// SIMATIC STEP 7 (V5.x) project e121001V002
// CPU: CPU 313C-2 DP
// CPU: CPU 313C-2 DP
// station: P_ADR_BUS
// station: Hardware
// station: OLD
// station: P_ADR_BUS
// station: Hardware
// station: SIMATIC 300(2)
// program: Programa S7(1)
// program: Programa S7(2)

SYMBOL_TABLE
"COUNT"	SFB 47	SFB 47	// Common counter module
"VAT_1"	VAT 1	
END_SYMBOL_TABLE

FUNCTION_BLOCK FB 30
VERSION : 0.1
BEGIN
// (block stored without names or comments; labels and parameter names are numbered)
NETWORK
TITLE =
      A     M 251.0;
      =     L 16.0;
      A     L 16.0;
      JNB   M001;
      L     DIW [AR2,P#26.0];
      L     DIW [AR2,P#4.0];
      +I;
      T     DIW [AR2,P#28.0];
M001: NOP   0;
      A     L 16.0;
      A(;
      A(;
      L     DID [AR2,P#0.0];
      L     DIW [AR2,P#26.0];
      >=I;
      );
      A(;
      L     DID [AR2,P#0.0];
      L     DIW [AR2,P#36.0];
      <I;
      );
      O;
      A(;
      L     DID [AR2,P#0.0];
      L     DIW [AR2,P#26.0];
      >=I;
      );
      A(;
      L     DID [AR2,P#0.0];
      L     DIW [AR2,P#28.0];
      <I;
      );
      );
      =     DIX [AR2,P#16.0];
NETWORK
TITLE =
      A     DIX [AR2,P#16.0];
      =     L 16.0;
      A     L 16.0;
      JNB   M002;
      L     DIW [AR2,P#34.0];
      L     164;
      *I;
      T     DIW [AR2,P#14.0];
M002: NOP   0;
      A     L 16.0;
      JNB   M003;
      L     0;
      T     DIW [AR2,P#18.0];
M003: NOP   0;
NETWORK
TITLE =
      A     M 251.0;
      =     L 16.0;
      A     L 16.0;
      JNB   M004;
      L     DIW [AR2,P#36.0];
      L     DIW [AR2,P#4.0];
      +I;
      T     DIW [AR2,P#38.0];
M004: NOP   0;
      A     L 16.0;
      A(;
      A(;
      L     DID [AR2,P#0.0];
      L     DIW [AR2,P#36.0];
      >=I;
      );
      A(;
      L     DID [AR2,P#0.0];
      L     DIW [AR2,P#46.0];
      <I;
      );
      O;
      A(;
      L     DID [AR2,P#0.0];
      L     DIW [AR2,P#36.0];
      >=I;
      );
      A(;
      L     DID [AR2,P#0.0];
      L     DIW [AR2,P#38.0];
      <I;
      );
      );
      =     DIX [AR2,P#16.1];
NETWORK
TITLE =
      A     DIX [AR2,P#16.1];
      =     L 16.0;
      A     L 16.0;
      AN    T 13;
      =     L 16.1;
      A     L 16.1;
      JNB   M005;
      L     DIW [AR2,P#44.0];
      L     164;
      *I;
      T     DIW [AR2,P#14.0];
M005: NOP   0;
      A     L 16.1;
      JNB   M006;
      L     1;
      T     DIW [AR2,P#18.0];
M006: NOP   0;
      A     L 16.0;
      A     T 13;
      =     L 16.1;
      A     L 16.1;
      JNB   M007;
      L     80;
      L     164;
      *I;
      T     DIW [AR2,P#14.0];
M007: NOP   0;
      A     L 16.1;
      JNB   M008;
      L     1;
      T     DIW [AR2,P#18.0];
M008: NOP   0;
NETWORK
TITLE =
      A     M 251.0;
      =     L 16.0;
      A     L 16.0;
      JNB   M009;
      L     DIW [AR2,P#46.0];
      L     DIW [AR2,P#4.0];
      +I;
      T     DIW [AR2,P#48.0];
M009: NOP   0;
      A     L 16.0;
      A(;
      A(;
      L     DID [AR2,P#0.0];
      L     DIW [AR2,P#46.0];
      >=I;
      );
      A(;
      L     DID [AR2,P#0.0];
      L     DIW [AR2,P#56.0];
      <I;
      );
      O;
      A(;
      L     DID [AR2,P#0.0];
      L     DIW [AR2,P#46.0];
      >=I;
      );
      A(;
      L     DID [AR2,P#0.0];
      L     DIW [AR2,P#48.0];
      <I;
      );
      );
      =     DIX [AR2,P#16.2];
NETWORK
TITLE =
      A     DIX [AR2,P#16.2];
      =     L 16.0;
      A     L 16.0;
      AN    T 13;
      =     L 16.1;
      A     L 16.1;
      JNB   M010;
      L     DIW [AR2,P#54.0];
      L     164;
      *I;
      T     DIW [AR2,P#14.0];
M010: NOP   0;
      A     L 16.1;
      JNB   M011;
      L     2;
      T     DIW [AR2,P#18.0];
M011: NOP   0;
      A     L 16.0;
      A     T 13;
      =     L 16.1;
      A     L 16.1;
      JNB   M012;
      L     80;
      L     164;
      *I;
      T     DIW [AR2,P#14.0];
M012: NOP   0;
      A     L 16.1;
      JNB   M013;
      L     1;
      T     DIW [AR2,P#18.0];
M013: NOP   0;
NETWORK
TITLE =
      A     M 251.0;
      =     L 16.0;
      A     L 16.0;
      JNB   M014;
      L     DIW [AR2,P#56.0];
      L     DIW [AR2,P#4.0];
      +I;
      T     DIW [AR2,P#58.0];
M014: NOP   0;
      A     L 16.0;
      A(;
      A(;
      L     DID [AR2,P#0.0];
      L     DIW [AR2,P#56.0];
      >=I;
      );
      A(;
      L     DID [AR2,P#0.0];
      L     DIW [AR2,P#66.0];
      <I;
      );
      O;
      A(;
      L     DID [AR2,P#0.0];
      L     DIW [AR2,P#56.0];
      >=I;
      );
      A(;
      L     DID [AR2,P#0.0];
      L     DIW [AR2,P#58.0];
      <I;
      );
      );
      =     DIX [AR2,P#16.3];
NETWORK
TITLE =
      A     DIX [AR2,P#16.3];
      =     L 16.0;
      A     L 16.0;
      AN    T 13;
      =     L 16.1;
      A     L 16.1;
      JNB   M015;
      L     DIW [AR2,P#64.0];
      L     164;
      *I;
      T     DIW [AR2,P#14.0];
M015: NOP   0;
      A     L 16.1;
      JNB   M016;
      L     3;
      T     DIW [AR2,P#18.0];
M016: NOP   0;
      A     L 16.0;
      A     T 13;
      =     L 16.1;
      A     L 16.1;
      JNB   M017;
      L     80;
      L     164;
      *I;
      T     DIW [AR2,P#14.0];
M017: NOP   0;
      A     L 16.1;
      JNB   M018;
      L     3;
      T     DIW [AR2,P#18.0];
M018: NOP   0;
NETWORK
TITLE =
      A     M 251.0;
      =     L 16.0;
      A     L 16.0;
      JNB   M019;
      L     DIW [AR2,P#66.0];
      L     DIW [AR2,P#4.0];
      +I;
      T     DIW [AR2,P#68.0];
M019: NOP   0;
      A     L 16.0;
      A(;
      A(;
      L     DID [AR2,P#0.0];
      L     DIW [AR2,P#66.0];
      >=I;
      );
      A(;
      L     DID [AR2,P#0.0];
      L     DIW [AR2,P#76.0];
      <I;
      );
      O;
      A(;
      L     DID [AR2,P#0.0];
      L     DIW [AR2,P#66.0];
      >=I;
      );
      A(;
      L     DID [AR2,P#0.0];
      L     DIW [AR2,P#68.0];
      <I;
      );
      );
      =     DIX [AR2,P#16.4];
NETWORK
TITLE =
      A     DIX [AR2,P#16.4];
      =     L 16.0;
      A     L 16.0;
      AN    T 13;
      =     L 16.1;
      A     L 16.1;
      JNB   M020;
      L     DIW [AR2,P#74.0];
      L     164;
      *I;
      T     DIW [AR2,P#14.0];
M020: NOP   0;
      A     L 16.1;
      JNB   M021;
      L     4;
      T     DIW [AR2,P#18.0];
M021: NOP   0;
      A     L 16.0;
      A     T 13;
      =     L 16.1;
      A     L 16.1;
      JNB   M022;
      L     80;
      L     164;
      *I;
      T     DIW [AR2,P#14.0];
M022: NOP   0;
      A     L 16.1;
      JNB   M023;
      L     4;
      T     DIW [AR2,P#18.0];
M023: NOP   0;
NETWORK
TITLE =
      A     M 251.0;
      =     L 16.0;
      A     L 16.0;
      JNB   M024;
      L     DIW [AR2,P#76.0];
      L     DIW [AR2,P#4.0];
      +I;
      T     DIW [AR2,P#78.0];
M024: NOP   0;
      A     L 16.0;
      A(;
      A(;
      L     DID [AR2,P#0.0];
      L     DIW [AR2,P#76.0];
      >=I;
      );
      A(;
      L     DID [AR2,P#0.0];
      L     DIW [AR2,P#86.0];
      <I;
      );
      O;
      A(;
      L     DID [AR2,P#0.0];
      L     DIW [AR2,P#76.0];
      >=I;
      );
      A(;
      L     DID [AR2,P#0.0];
      L     DIW [AR2,P#78.0];
      <I;
      );
      );
      =     DIX [AR2,P#16.5];
NETWORK
TITLE =
      A     DIX [AR2,P#16.5];
      =     L 16.0;
      A     L 16.0;
      AN    T 13;
      =     L 16.1;
      A     L 16.1;
      JNB   M025;
      L     DIW [AR2,P#84.0];
      L     164;
      *I;
      T     DIW [AR2,P#14.0];
M025: NOP   0;
      A     L 16.1;
      JNB   M026;
      L     5;
      T     DIW [AR2,P#18.0];
M026: NOP   0;
      A     L 16.0;
      A     T 13;
      =     L 16.1;
      A     L 16.1;
      JNB   M027;
      L     80;
      L     164;
      *I;
      T     DIW [AR2,P#14.0];
M027: NOP   0;
      A     L 16.1;
      JNB   M028;
      L     5;
      T     DIW [AR2,P#18.0];
M028: NOP   0;
NETWORK
TITLE =
      A     M 251.0;
      =     L 16.0;
      A     L 16.0;
      JNB   M029;
      L     DIW [AR2,P#86.0];
      L     DIW [AR2,P#4.0];
      +I;
      T     DIW [AR2,P#88.0];
M029: NOP   0;
      A     L 16.0;
      A(;
      A(;
      L     DID [AR2,P#0.0];
      L     DIW [AR2,P#86.0];
      >=I;
      );
      A(;
      L     DID [AR2,P#0.0];
      L     DIW [AR2,P#96.0];
      <I;
      );
      O;
      A(;
      L     DID [AR2,P#0.0];
      L     DIW [AR2,P#86.0];
      >=I;
      );
      A(;
      L     DID [AR2,P#0.0];
      L     DIW [AR2,P#88.0];
      <I;
      );
      );
      =     DIX [AR2,P#16.6];
NETWORK
TITLE =
      A     DIX [AR2,P#16.6];
      =     L 16.0;
      A     L 16.0;
      AN    T 13;
      =     L 16.1;
      A     L 16.1;
      JNB   M030;
      L     DIW [AR2,P#94.0];
      L     164;
      *I;
      T     DIW [AR2,P#14.0];
M030: NOP   0;
      A     L 16.1;
      JNB   M031;
      L     6;
      T     DIW [AR2,P#18.0];
M031: NOP   0;
      A     L 16.0;
      A     T 13;
      =     L 16.1;
      A     L 16.1;
      JNB   M032;
      L     80;
      L     164;
      *I;
      T     DIW [AR2,P#14.0];
M032: NOP   0;
      A     L 16.1;
      JNB   M033;
      L     6;
      T     DIW [AR2,P#18.0];
M033: NOP   0;
NETWORK
TITLE =
      A     M 251.0;
      =     L 16.0;
      A     L 16.0;
      JNB   M034;
      L     DIW [AR2,P#96.0];
      L     DIW [AR2,P#4.0];
      +I;
      T     DIW [AR2,P#98.0];
M034: NOP   0;
      A     L 16.0;
      A(;
      A(;
      L     DID [AR2,P#0.0];
      L     DIW [AR2,P#96.0];
      >=I;
      );
      A(;
      L     DID [AR2,P#0.0];
      L     DIW [AR2,P#106.0];
      <I;
      );
      O;
      A(;
      L     DID [AR2,P#0.0];
      L     DIW [AR2,P#96.0];
      >=I;
      );
      A(;
      L     DID [AR2,P#0.0];
      L     DIW [AR2,P#98.0];
      <I;
      );
      );
      =     DIX [AR2,P#16.7];
NETWORK
TITLE =
      A     DIX [AR2,P#16.7];
      =     L 16.0;
      A     L 16.0;
      AN    T 13;
      =     L 16.1;
      A     L 16.1;
      JNB   M035;
      L     DIW [AR2,P#104.0];
      L     164;
      *I;
      T     DIW [AR2,P#14.0];
M035: NOP   0;
      A     L 16.1;
      JNB   M036;
      L     7;
      T     DIW [AR2,P#18.0];
M036: NOP   0;
      A     L 16.0;
      A     T 13;
      =     L 16.1;
      A     L 16.1;
      JNB   M037;
      L     80;
      L     164;
      *I;
      T     DIW [AR2,P#14.0];
M037: NOP   0;
      A     L 16.1;
      JNB   M038;
      L     7;
      T     DIW [AR2,P#18.0];
M038: NOP   0;
NETWORK
TITLE =
      A     M 251.0;
      =     L 16.0;
      A     L 16.0;
      JNB   M039;
      L     DIW [AR2,P#106.0];
      L     DIW [AR2,P#4.0];
      +I;
      T     DIW [AR2,P#108.0];
M039: NOP   0;
      A     L 16.0;
      A(;
      L     DID [AR2,P#0.0];
      L     DIW [AR2,P#106.0];
      >=I;
      );
      A(;
      L     DID [AR2,P#0.0];
      L     DIW [AR2,P#108.0];
      <I;
      );
      =     DIX [AR2,P#17.0];
NETWORK
TITLE =
      A     DIX [AR2,P#17.0];
      =     L 16.0;
      A     L 16.0;
      JNB   M040;
      L     DIW [AR2,P#114.0];
      L     164;
      *I;
      T     DIW [AR2,P#14.0];
M040: NOP   0;
      A     L 16.0;
      JNB   M041;
      L     8;
      T     DIW [AR2,P#18.0];
M041: NOP   0;
NETWORK
TITLE =
      A     DIX [AR2,P#8.0];
      =     L 26.0;
      A     L 26.0;
      JNB   M042;
      L     DIW [AR2,P#6.0];
      L     5;
      *I;
      T     LW 2;
M042: NOP   0;
      A     L 26.0;
      JNB   M043;
      L     LW 2;
      L     13;
      +I;
      T     LW 4;
M043: NOP   0;
      A     L 26.0;
      JNB   M044;
      CALL  FC 103 (
           $1                       := 30,
           $2                       := 1,
           $3                       := 1,
           $4                       := 30,
           $5                       := P#L 4.0);
M044: NOP   0;
      A     L 26.0;
      JNB   M045;
      L     LW 2;
      L     17;
      +I;
      T     LW 6;
M045: NOP   0;
      A     L 26.0;
      JNB   M046;
      CALL  FC 103 (
           $1                       := 30,
           $2                       := 12,
           $3                       := 12,
           $4                       := 30,
           $5                       := P#L 6.0);
M046: NOP   0;
      A     L 26.0;
      JNB   M047;
      L     DIW [AR2,P#22.0];
      L     100;
      +I;
      T     LW 0;
M047: NOP   0;
      A     L 26.0;
      JNB   M048;
      CALL  FC 103 (
           $1                       := 30,
           $2                       := 13,
           $3                       := 92,
           $4                       := P#L 0.0,
           $5                       := 2);
M048: NOP   0;
      A     L 26.0;
      BLD   102;
      R     DB30.DBX 8.0;
      A(;
      A     L 26.0;
      JNB   M049;
      L     DB30.DBW 6;
      L     1;
      +I;
      T     DB30.DBW 6;
      AN    OV;
      SAVE;
      CLR;
M049: A     BR;
      );
      A(;
      L     DB30.DBW 6;
      L     8;
      >I;
      );
      JNB   M050;
      L     8;
      T     DB30.DBW 6;
M050: NOP   0;
NETWORK
TITLE =
      A     DIX [AR2,P#8.1];
      =     L 26.0;
      A     L 26.0;
      JNB   M051;
      L     DIW [AR2,P#6.0];
      L     5;
      *I;
      T     LW 2;
M051: NOP   0;
      A     L 26.0;
      JNB   M052;
      L     LW 2;
      L     17;
      +I;
      T     LW 4;
M052: NOP   0;
      A     L 26.0;
      JNB   M053;
      CALL  FC 103 (
           $1                       := 30,
           $2                       := 12,
           $3                       := 12,
           $4                       := 30,
           $5                       := P#L 4.0);
M053: NOP   0;
      A     L 26.0;
      JNB   M054;
      L     DIW [AR2,P#22.0];
      L     100;
      +I;
      T     LW 0;
M054: NOP   0;
      A     L 26.0;
      JNB   M055;
      CALL  FC 103 (
           $1                       := 30,
           $2                       := 13,
           $3                       := 92,
           $4                       := P#L 0.0,
           $5                       := 2);
M055: NOP   0;
      A     L 26.0;
      BLD   102;
      R     DB30.DBX 8.1;
NETWORK
TITLE =
      A     DIX [AR2,P#8.4];
      =     L 26.0;
      A     L 26.0;
      JNB   M056;
      L     DIW [AR2,P#22.0];
      L     100;
      +I;
      T     LW 0;
M056: NOP   0;
      A     L 26.0;
      JNB   M057;
      CALL  FC 103 (
           $1                       := 30,
           $2                       := 13,
           $3                       := 92,
           $4                       := P#L 0.0,
           $5                       := 2);
M057: NOP   0;
      A     L 26.0;
      BLD   102;
      R     M 4.0;
NETWORK
TITLE =
      A     DIX [AR2,P#8.5];
      =     L 26.0;
      A     L 26.0;
      JNB   M058;
      L     DB1.DBW 42;
      L     100;
      +I;
      T     LW 8;
M058: NOP   0;
      A     L 26.0;
      JNB   M059;
      CALL  FC 103 (
           $1                       := 121,
           $2                       := 2,
           $3                       := 92,
           $4                       := P#L 8.0,
           $5                       := 2);
M059: NOP   0;
      A     L 26.0;
      BLD   102;
      R     M 4.2;
NETWORK
TITLE =
      A     DIX [AR2,P#8.3];
      =     L 26.0;
      A     L 26.0;
      JNB   M060;
      L     DB1.DBW 38;
      L     100;
      +I;
      T     LW 10;
M060: NOP   0;
      A     L 26.0;
      JNB   M061;
      L     DB1.DBW 40;
      L     100;
      +I;
      T     LW 12;
M061: NOP   0;
      A     L 26.0;
      JNB   M062;
      CALL  FC 103 (
           $1                       := P#L 10.0,
           $2                       := 2,
           $3                       := 92,
           $4                       := P#L 12.0,
           $5                       := 2);
M062: NOP   0;
      A     L 26.0;
      BLD   102;
      R     M 4.1;
NETWORK
TITLE =
      A     DIX [AR2,P#8.6];
      =     L 26.0;
      A     L 26.0;
      JNB   M063;
      L     DB1.DBW 12;
      L     77;
      +I;
      T     LW 14;
M063: NOP   0;
      A     L 26.0;
      JNB   M064;
      CALL  FC 103 (
           $1                       := 30,
           $2                       := 6,
           $3                       := 6,
           $4                       := 30,
           $5                       := P#L 14.0);
M064: NOP   0;
      A     L 26.0;
      JNB   M065;
      L     DIW [AR2,P#22.0];
      L     100;
      +I;
      T     LW 0;
M065: NOP   0;
      A     L 26.0;
      JNB   M066;
      CALL  FC 103 (
           $1                       := 30,
           $2                       := 13,
           $3                       := 92,
           $4                       := P#L 0.0,
           $5                       := 2);
M066: NOP   0;
      A     L 26.0;
      BLD   102;
      R     DB30.DBX 8.6;
      A(;
      A     L 26.0;
      JNB   M067;
      L     DB1.DBW 12;
      L     1;
      +I;
      T     DB1.DBW 12;
      AN    OV;
      SAVE;
      CLR;
M067: A     BR;
      );
      A(;
      L     DB1.DBW 12;
      L     3;
      >I;
      );
      JNB   M068;
      L     3;
      T     DB1.DBW 12;
M068: NOP   0;
NETWORK
TITLE =
      A     M 251.0;
      =     L 26.0;
      A     L 26.0;
      JNB   M069;
      L     DIW [AR2,P#154.0];
      L     10;
      +I;
      T     DIW [AR2,P#166.0];
M069: NOP   0;
      A     L 26.0;
      JNB   M070;
      L     DIW [AR2,P#154.0];
      L     10;
      -I;
      T     DIW [AR2,P#168.0];
M070: NOP   0;
      A     L 26.0;
      A(;
      L     DIW [AR2,P#12.0];
      L     DIW [AR2,P#168.0];
      >=I;
      );
      A(;
      L     DIW [AR2,P#12.0];
      L     DIW [AR2,P#166.0];
      <=I;
      );
      =     DIX [AR2,P#20.0];
NETWORK
TITLE =
      A     M 251.0;
      =     L 26.0;
      A     L 26.0;
      JNB   M071;
      L     DIW [AR2,P#156.0];
      L     10;
      +I;
      T     DIW [AR2,P#170.0];
M071: NOP   0;
      A     L 26.0;
      JNB   M072;
      L     DIW [AR2,P#156.0];
      L     10;
      -I;
      T     LW 16;
M072: NOP   0;
      A     L 26.0;
      A(;
      L     DIW [AR2,P#12.0];
      L     LW 16;
      >=I;
      );
      A(;
      L     DIW [AR2,P#12.0];
      L     DIW [AR2,P#170.0];
      <=I;
      );
      =     DIX [AR2,P#20.1];
NETWORK
TITLE =
      A     M 251.0;
      =     L 26.0;
      A     L 26.0;
      JNB   M073;
      L     DIW [AR2,P#158.0];
      L     10;
      +I;
      T     LW 18;
M073: NOP   0;
      A     L 26.0;
      JNB   M074;
      L     DIW [AR2,P#158.0];
      L     10;
      -I;
      T     LW 20;
M074: NOP   0;
      A     L 26.0;
      A(;
      L     DIW [AR2,P#12.0];
      L     LW 20;
      >=I;
      );
      A(;
      L     DIW [AR2,P#12.0];
      L     LW 18;
      <=I;
      );
      =     DIX [AR2,P#20.2];
NETWORK
TITLE =
      A     M 251.0;
      =     L 26.0;
      A     L 26.0;
      JNB   M075;
      L     DIW [AR2,P#160.0];
      L     10;
      +I;
      T     LW 22;
M075: NOP   0;
      A     L 26.0;
      JNB   M076;
      L     DIW [AR2,P#160.0];
      L     10;
      -I;
      T     LW 24;
M076: NOP   0;
      A     L 26.0;
      A(;
      L     DIW [AR2,P#12.0];
      L     LW 24;
      >=I;
      );
      A(;
      L     DIW [AR2,P#12.0];
      L     LW 22;
      <=I;
      );
      =     DIX [AR2,P#20.3];
NETWORK
TITLE =
      A     M 80.0;
      A     DIX [AR2,P#20.0];
      =     M 6.5;
END_FUNCTION_BLOCK

FUNCTION_BLOCK FB 50
VERSION : 0.1
BEGIN
// (block stored without names or comments; labels and parameter names are numbered)
NETWORK
TITLE =
END_FUNCTION_BLOCK

FUNCTION_BLOCK FB 51
VERSION : 0.1
BEGIN
// (block stored without names or comments; labels and parameter names are numbered)
NETWORK
TITLE =
END_FUNCTION_BLOCK

FUNCTION FC 1 : VOID
VERSION : 0.1
BEGIN
// (block stored without names or comments; labels and parameter names are numbered)
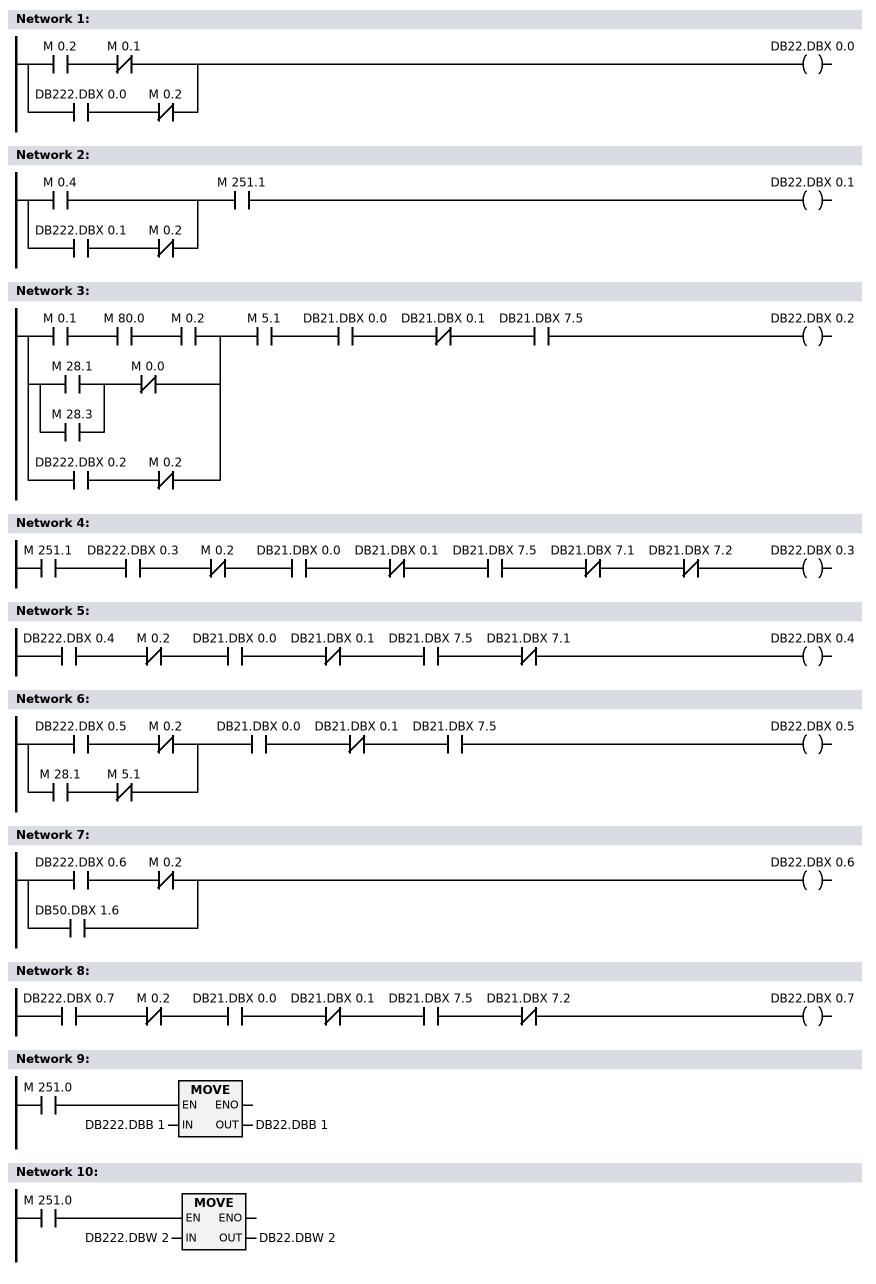
NETWORK
TITLE =
      A     M 0.2;
      AN    M 0.1;
      O;
      A     DB222.DBX 0.0;
      AN    M 0.2;
      =     DB22.DBX 0.0;
NETWORK
TITLE =
      A(;
      O     M 0.4;
      O;
      A     DB222.DBX 0.1;
      AN    M 0.2;
      );
      A     M 251.1;
      =     DB22.DBX 0.1;
NETWORK
TITLE =
      A(;
      A     M 0.1;
      A     M 80.0;
      A     M 0.2;
      O;
      A(;
      O     M 28.1;
      O     M 28.3;
      );
      AN    M 0.0;
      O;
      A     DB222.DBX 0.2;
      AN    M 0.2;
      );
      A     M 5.1;
      A     DB21.DBX 0.0;
      AN    DB21.DBX 0.1;
      A     DB21.DBX 7.5;
      =     DB22.DBX 0.2;
NETWORK
TITLE =
      A     M 251.1;
      A     DB222.DBX 0.3;
      AN    M 0.2;
      A     DB21.DBX 0.0;
      AN    DB21.DBX 0.1;
      A     DB21.DBX 7.5;
      AN    DB21.DBX 7.1;
      AN    DB21.DBX 7.2;
      =     DB22.DBX 0.3;
NETWORK
TITLE =
      A     DB222.DBX 0.4;
      AN    M 0.2;
      A     DB21.DBX 0.0;
      AN    DB21.DBX 0.1;
      A     DB21.DBX 7.5;
      AN    DB21.DBX 7.1;
      =     DB22.DBX 0.4;
NETWORK
TITLE =
      A(;
      A     DB222.DBX 0.5;
      AN    M 0.2;
      O;
      A     M 28.1;
      AN    M 5.1;
      );
      A     DB21.DBX 0.0;
      AN    DB21.DBX 0.1;
      A     DB21.DBX 7.5;
      =     DB22.DBX 0.5;
NETWORK
TITLE =
      A     DB222.DBX 0.6;
      AN    M 0.2;
      O     DB50.DBX 1.6;
      =     DB22.DBX 0.6;
NETWORK
TITLE =
      A     DB222.DBX 0.7;
      AN    M 0.2;
      A     DB21.DBX 0.0;
      AN    DB21.DBX 0.1;
      A     DB21.DBX 7.5;
      AN    DB21.DBX 7.2;
      =     DB22.DBX 0.7;
NETWORK
TITLE =
      A     M 251.0;
      JNB   M001;
      L     DB222.DBB 1;
      T     DB22.DBB 1;
M001: NOP   0;
NETWORK
TITLE =
      A     M 251.0;
      JNB   M002;
      L     DB222.DBW 2;
      T     DB22.DBW 2;
M002: NOP   0;
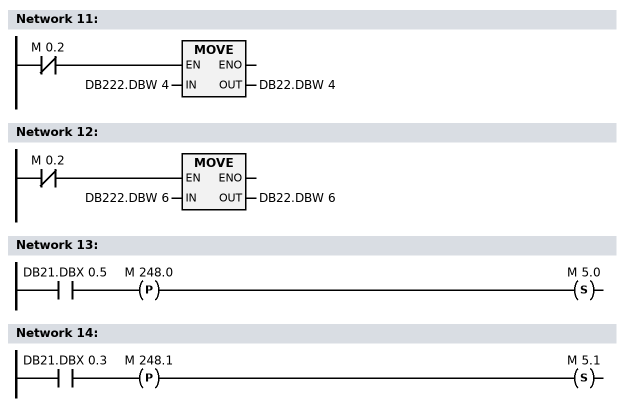
NETWORK
TITLE =
      AN    M 0.2;
      JNB   M003;
      L     DB222.DBW 4;
      T     DB22.DBW 4;
M003: NOP   0;
NETWORK
TITLE =
      AN    M 0.2;
      JNB   M004;
      L     DB222.DBW 6;
      T     DB22.DBW 6;
M004: NOP   0;
NETWORK
TITLE =
      A     DB21.DBX 0.5;
      FP    M 248.0;
      S     M 5.0;
NETWORK
TITLE =
      A     DB21.DBX 0.3;
      FP    M 248.1;
      S     M 5.1;
END_FUNCTION

FUNCTION FC 10 : VOID
VERSION : 0.1
VAR_TEMP
  TEMP0 : INT ;
END_VAR
BEGIN
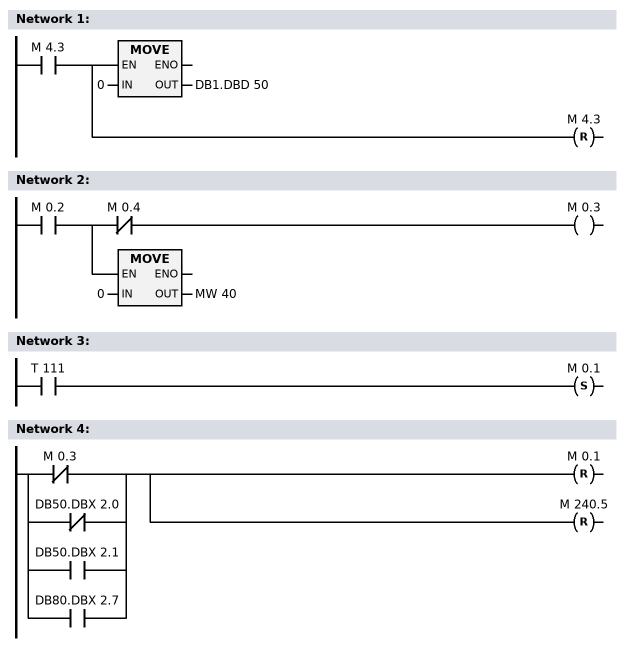
NETWORK
TITLE =
      A     M 4.3;
      =     L 2.0;
      A     L 2.0;
      JNB   _001;
      L     0;
      T     DB1.DBD 50;
_001: NOP   0;
      A     L 2.0;
      BLD   102;
      R     M 4.3;
NETWORK
TITLE =
      A     M 0.2;
      =     L 2.0;
      A     L 2.0;
      AN    M 0.4;
      =     M 0.3;
      A     L 2.0;
      JNB   _002;
      L     0;
      T     MW 40;
_002: NOP   0;
NETWORK
TITLE =
      A     T 111;
      S     M 0.1;
NETWORK
TITLE =
      ON    M 0.3;
      ON    DB50.DBX 2.0;
      O     DB50.DBX 2.1;
      O     DB80.DBX 2.7;
      R     M 0.1;
      R     M 240.5;
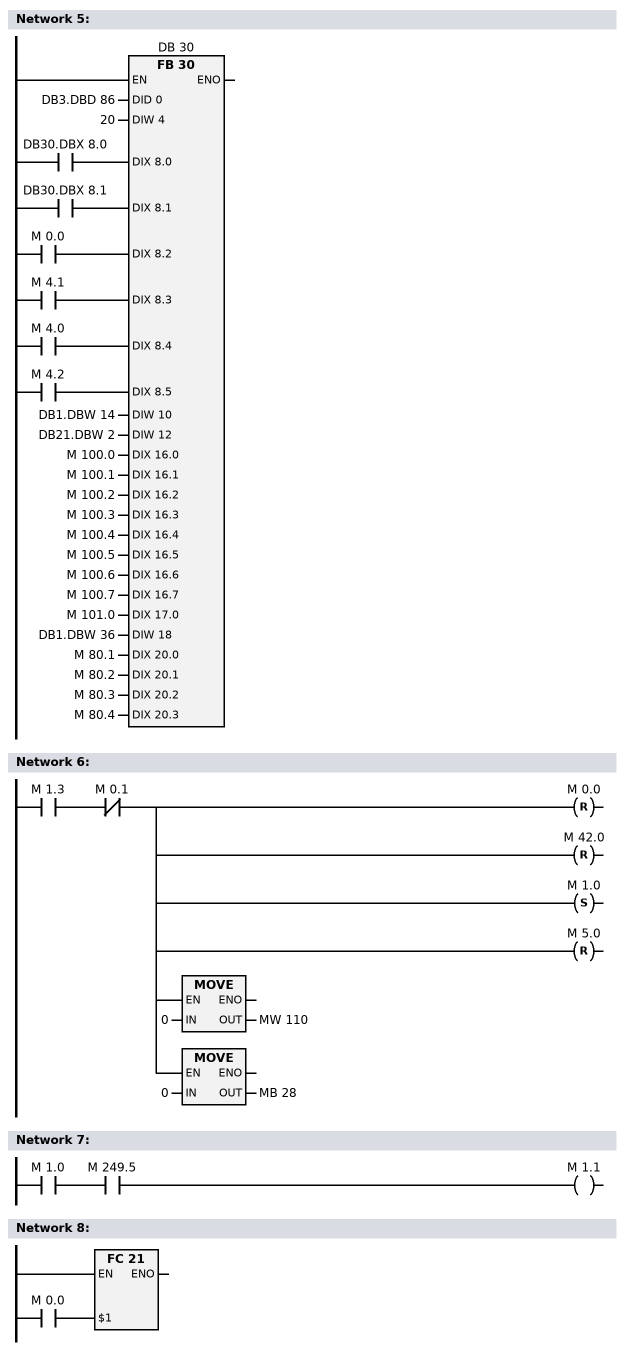
NETWORK
TITLE =
      A     DB30.DBX 8.0;
      =     L 2.0;
      BLD   103;
      A     DB30.DBX 8.1;
      =     L 2.1;
      BLD   103;
      A     M 0.0;
      =     L 2.2;
      BLD   103;
      A     M 4.1;
      =     L 2.3;
      BLD   103;
      A     M 4.0;
      =     L 2.4;
      BLD   103;
      A     M 4.2;
      =     L 2.5;
      BLD   103;
      CALL  FB 30 , DB 30 (
           DID 0                    := DB3.DBD 86,
           DIW 4                    := 20,
           DIX 8.0                  := L 2.0,
           DIX 8.1                  := L 2.1,
           DIX 8.2                  := L 2.2,
           DIX 8.3                  := L 2.3,
           DIX 8.4                  := L 2.4,
           DIX 8.5                  := L 2.5,
           DIW 10                   := DB1.DBW 14,
           DIW 12                   := DB21.DBW 2,
           DIX 16.0                 := M 100.0,
           DIX 16.1                 := M 100.1,
           DIX 16.2                 := M 100.2,
           DIX 16.3                 := M 100.3,
           DIX 16.4                 := M 100.4,
           DIX 16.5                 := M 100.5,
           DIX 16.6                 := M 100.6,
           DIX 16.7                 := M 100.7,
           DIX 17.0                 := M 101.0,
           DIW 18                   := DB1.DBW 36,
           DIX 20.0                 := M 80.1,
           DIX 20.1                 := M 80.2,
           DIX 20.2                 := M 80.3,
           DIX 20.3                 := M 80.4);
      NOP   0;
NETWORK
TITLE =
      A     M 1.3;
      AN    M 0.1;
      =     L 2.0;
      A     L 2.0;
      BLD   102;
      R     M 0.0;
      A     L 2.0;
      BLD   102;
      R     M 42.0;
      A     L 2.0;
      BLD   102;
      S     M 1.0;
      A     L 2.0;
      BLD   102;
      R     M 5.0;
      A     L 2.0;
      JNB   _003;
      L     0;
      T     MW 110;
_003: NOP   0;
      A     L 2.0;
      JNB   _004;
      L     0;
      T     MB 28;
_004: NOP   0;
NETWORK
TITLE =
      A     M 1.0;
      A     M 249.5;
      =     M 1.1;
NETWORK
TITLE =
      A     M 0.0;
      =     L 2.0;
      BLD   103;
      CALL  FC 21 (
           $1                       := L 2.0);
      NOP   0;
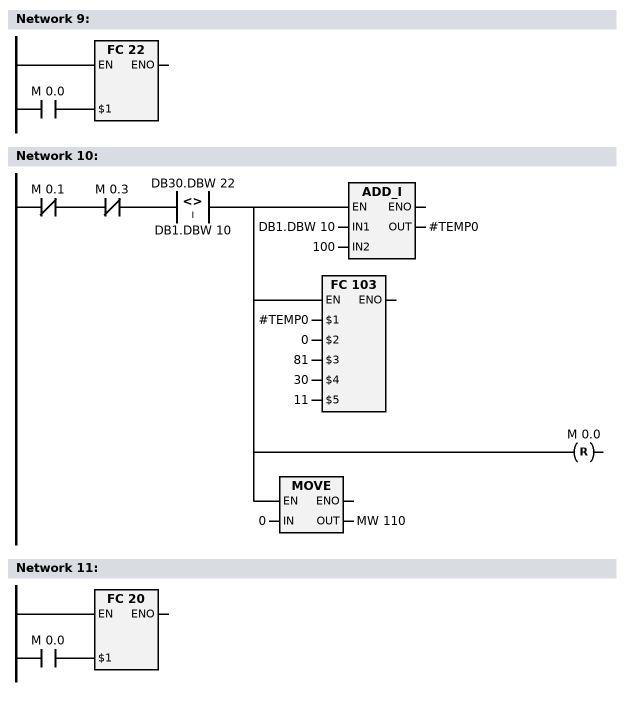
NETWORK
TITLE =
      A     M 0.0;
      =     L 2.0;
      BLD   103;
      CALL  FC 22 (
           $1                       := L 2.0);
      NOP   0;
NETWORK
TITLE =
      AN    M 0.1;
      AN    M 0.3;
      A(;
      L     DB30.DBW 22;
      L     DB1.DBW 10;
      <>I;
      );
      =     L 2.0;
      A     L 2.0;
      JNB   _005;
      L     DB1.DBW 10;
      L     100;
      +I;
      T     #TEMP0;
_005: NOP   0;
      A     L 2.0;
      JNB   _006;
      CALL  FC 103 (
           $1                       := #TEMP0,
           $2                       := 0,
           $3                       := 81,
           $4                       := 30,
           $5                       := 11);
_006: NOP   0;
      A     L 2.0;
      BLD   102;
      R     M 0.0;
      A     L 2.0;
      JNB   _007;
      L     0;
      T     MW 110;
_007: NOP   0;
NETWORK
TITLE =
      A     M 0.0;
      =     L 2.0;
      BLD   103;
      CALL  FC 20 (
           $1                       := L 2.0);
      NOP   0;
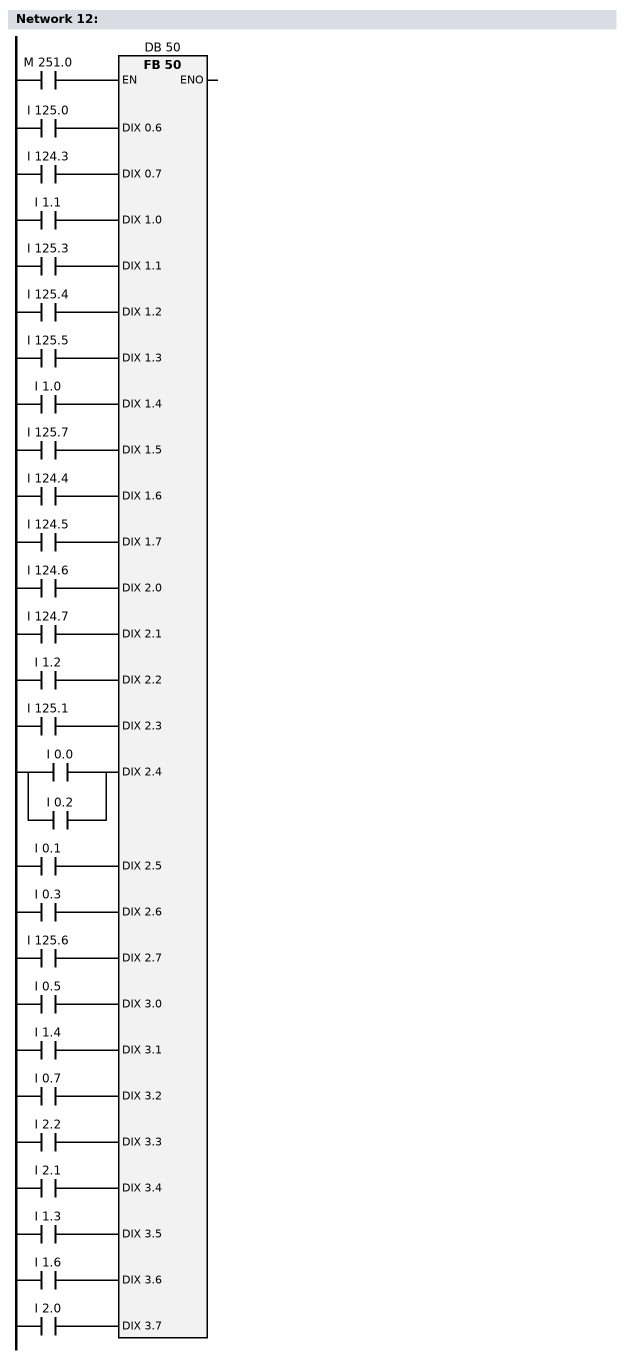
NETWORK
TITLE =
      A     I 125.0;
      =     L 2.6;
      BLD   103;
      A     I 124.3;
      =     L 2.7;
      BLD   103;
      A     I 1.1;
      =     L 3.0;
      BLD   103;
      A     I 125.3;
      =     L 3.1;
      BLD   103;
      A     I 125.4;
      =     L 3.2;
      BLD   103;
      A     I 125.5;
      =     L 3.3;
      BLD   103;
      A     I 1.0;
      =     L 3.4;
      BLD   103;
      A     I 125.7;
      =     L 3.5;
      BLD   103;
      A     I 124.4;
      =     L 3.6;
      BLD   103;
      A     I 124.5;
      =     L 3.7;
      BLD   103;
      A     I 124.6;
      =     L 4.0;
      BLD   103;
      A     I 124.7;
      =     L 4.1;
      BLD   103;
      A     I 1.2;
      =     L 4.2;
      BLD   103;
      A     I 125.1;
      =     L 4.3;
      BLD   103;
      A(;
      O     I 0.0;
      O     I 0.2;
      );
      =     L 4.4;
      BLD   103;
      A     I 0.1;
      =     L 4.5;
      BLD   103;
      A     I 0.3;
      =     L 4.6;
      BLD   103;
      A     I 125.6;
      =     L 4.7;
      BLD   103;
      A     I 0.5;
      =     L 5.0;
      BLD   103;
      A     I 1.4;
      =     L 5.1;
      BLD   103;
      A     I 0.7;
      =     L 5.2;
      BLD   103;
      A     I 2.2;
      =     L 5.3;
      BLD   103;
      A     I 2.1;
      =     L 5.4;
      BLD   103;
      A     I 1.3;
      =     L 5.5;
      BLD   103;
      A     I 1.6;
      =     L 5.6;
      BLD   103;
      A     I 2.0;
      =     L 5.7;
      BLD   103;
      A     M 251.0;
      JNB   _008;
      CALL  FB 50 , DB 50 (
           DIX 0.6                  := L 2.6,
           DIX 0.7                  := L 2.7,
           DIX 1.0                  := L 3.0,
           DIX 1.1                  := L 3.1,
           DIX 1.2                  := L 3.2,
           DIX 1.3                  := L 3.3,
           DIX 1.4                  := L 3.4,
           DIX 1.5                  := L 3.5,
           DIX 1.6                  := L 3.6,
           DIX 1.7                  := L 3.7,
           DIX 2.0                  := L 4.0,
           DIX 2.1                  := L 4.1,
           DIX 2.2                  := L 4.2,
           DIX 2.3                  := L 4.3,
           DIX 2.4                  := L 4.4,
           DIX 2.5                  := L 4.5,
           DIX 2.6                  := L 4.6,
           DIX 2.7                  := L 4.7,
           DIX 3.0                  := L 5.0,
           DIX 3.1                  := L 5.1,
           DIX 3.2                  := L 5.2,
           DIX 3.3                  := L 5.3,
           DIX 3.4                  := L 5.4,
           DIX 3.5                  := L 5.5,
           DIX 3.6                  := L 5.6,
           DIX 3.7                  := L 5.7);
_008: NOP   0;
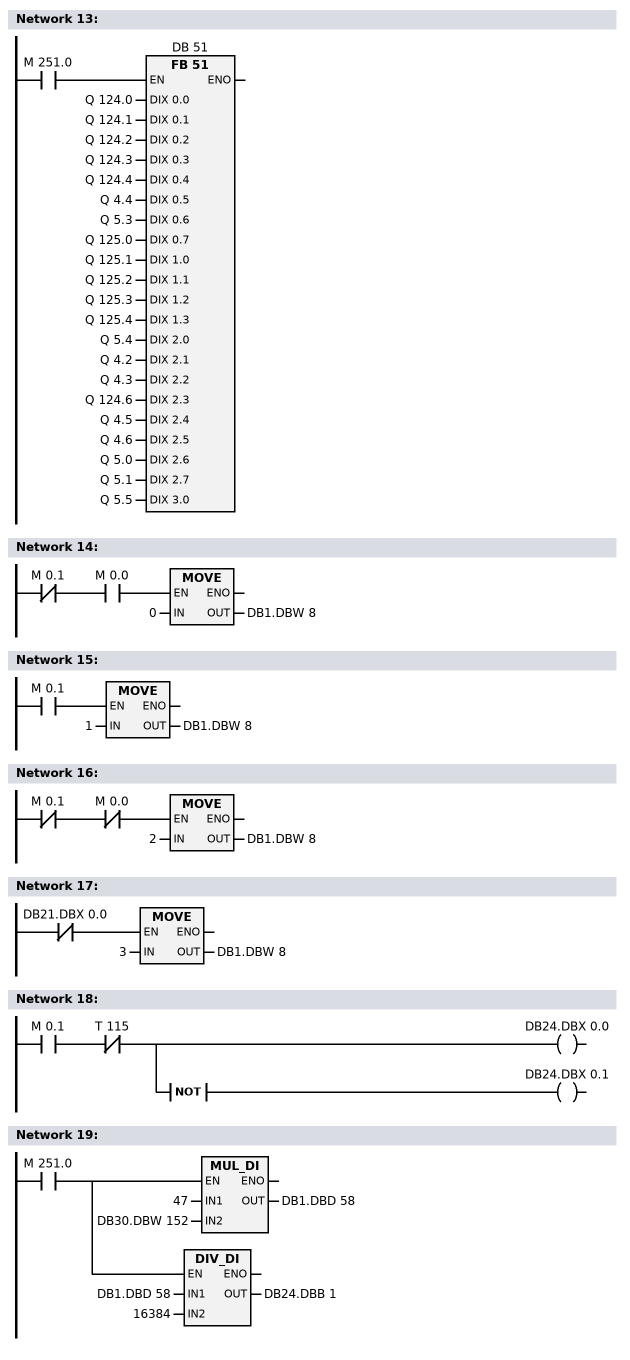
NETWORK
TITLE =
      A     M 251.0;
      JNB   _009;
      CALL  FB 51 , DB 51 (
           DIX 0.0                  := Q 124.0,
           DIX 0.1                  := Q 124.1,
           DIX 0.2                  := Q 124.2,
           DIX 0.3                  := Q 124.3,
           DIX 0.4                  := Q 124.4,
           DIX 0.5                  := Q 4.4,
           DIX 0.6                  := Q 5.3,
           DIX 0.7                  := Q 125.0,
           DIX 1.0                  := Q 125.1,
           DIX 1.1                  := Q 125.2,
           DIX 1.2                  := Q 125.3,
           DIX 1.3                  := Q 125.4,
           DIX 2.0                  := Q 5.4,
           DIX 2.1                  := Q 4.2,
           DIX 2.2                  := Q 4.3,
           DIX 2.3                  := Q 124.6,
           DIX 2.4                  := Q 4.5,
           DIX 2.5                  := Q 4.6,
           DIX 2.6                  := Q 5.0,
           DIX 2.7                  := Q 5.1,
           DIX 3.0                  := Q 5.5);
_009: NOP   0;
NETWORK
TITLE =
      AN    M 0.1;
      A     M 0.0;
      JNB   _00a;
      L     0;
      T     DB1.DBW 8;
_00a: NOP   0;
NETWORK
TITLE =
      A     M 0.1;
      JNB   _00b;
      L     1;
      T     DB1.DBW 8;
_00b: NOP   0;
NETWORK
TITLE =
      AN    M 0.1;
      AN    M 0.0;
      JNB   _00c;
      L     2;
      T     DB1.DBW 8;
_00c: NOP   0;
NETWORK
TITLE =
      AN    DB21.DBX 0.0;
      JNB   _00d;
      L     3;
      T     DB1.DBW 8;
_00d: NOP   0;
NETWORK
TITLE =
      A     M 0.1;
      AN    T 115;
      =     L 2.0;
      A     L 2.0;
      BLD   102;
      =     DB24.DBX 0.0;
      A     L 2.0;
      NOT;
      =     DB24.DBX 0.1;
NETWORK
TITLE =
      A     M 251.0;
      =     L 2.0;
      A     L 2.0;
      JNB   _00e;
      L     47;
      L     DB30.DBW 152;
      *D;
      T     DB1.DBD 58;
_00e: NOP   0;
      A     L 2.0;
      JNB   _00f;
      L     DB1.DBD 58;
      L     16384;
      /D;
      T     DB24.DBB 1;
_00f: NOP   0;
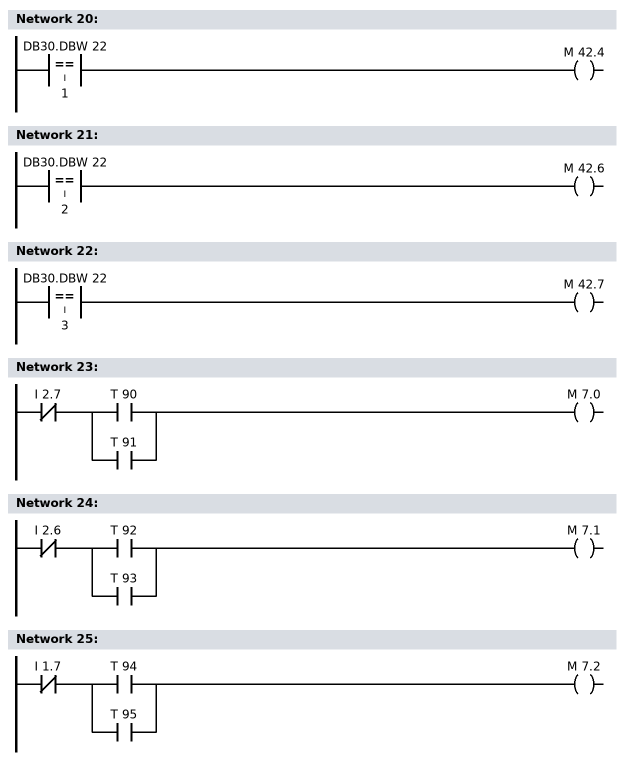
NETWORK
TITLE =
      L     DB30.DBW 22;
      L     1;
      ==I;
      =     M 42.4;
NETWORK
TITLE =
      L     DB30.DBW 22;
      L     2;
      ==I;
      =     M 42.6;
NETWORK
TITLE =
      L     DB30.DBW 22;
      L     3;
      ==I;
      =     M 42.7;
NETWORK
TITLE =
      AN    I 2.7;
      A(;
      O     T 90;
      O     T 91;
      );
      =     M 7.0;
NETWORK
TITLE =
      AN    I 2.6;
      A(;
      O     T 92;
      O     T 93;
      );
      =     M 7.1;
NETWORK
TITLE =
      AN    I 1.7;
      A(;
      O     T 94;
      O     T 95;
      );
      =     M 7.2;
END_FUNCTION

FUNCTION FC 18 : VOID
VERSION : 0.1
BEGIN
// (block stored without names or comments; labels and parameter names are numbered)
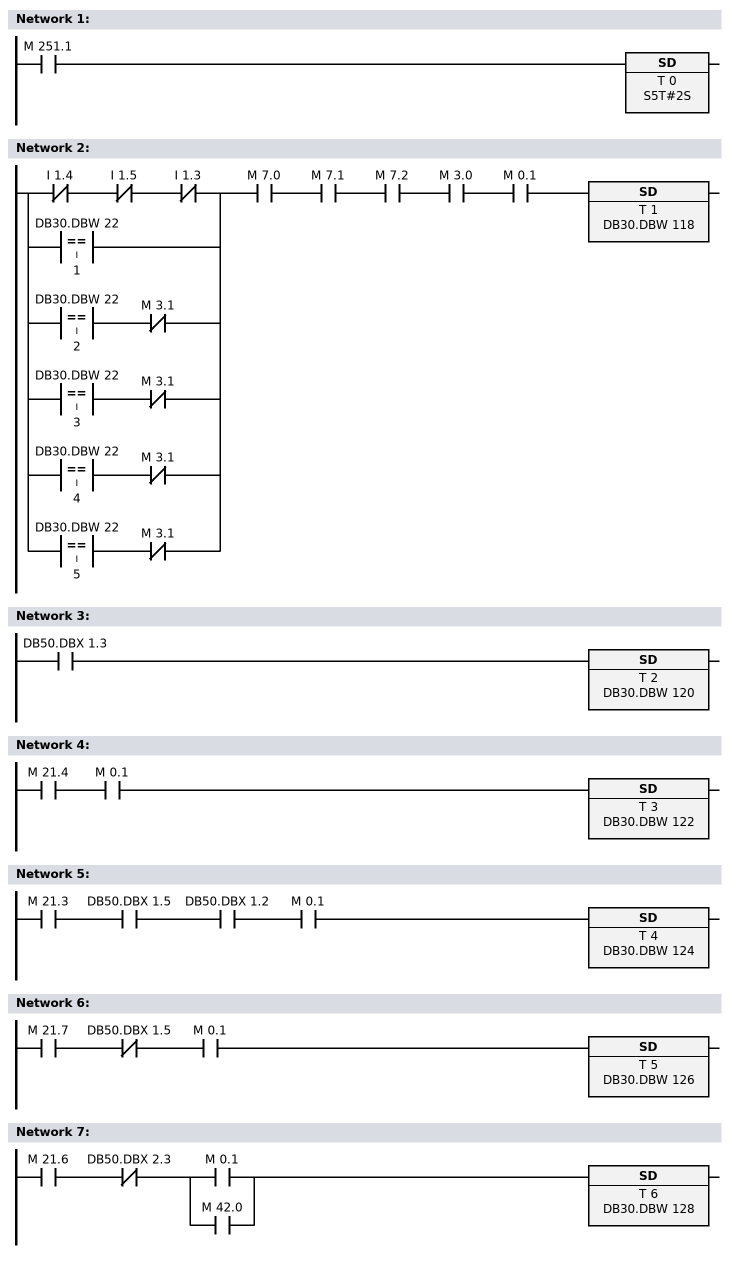
NETWORK
TITLE =
      A     M 251.1;
      L     S5T#2S;
      SD    T 0;
NETWORK
TITLE =
      A(;
      AN    I 1.4;
      AN    I 1.5;
      AN    I 1.3;
      O(;
      L     DB30.DBW 22;
      L     1;
      ==I;
      );
      O;
      A(;
      L     DB30.DBW 22;
      L     2;
      ==I;
      );
      AN    M 3.1;
      O;
      A(;
      L     DB30.DBW 22;
      L     3;
      ==I;
      );
      AN    M 3.1;
      O;
      A(;
      L     DB30.DBW 22;
      L     4;
      ==I;
      );
      AN    M 3.1;
      O;
      A(;
      L     DB30.DBW 22;
      L     5;
      ==I;
      );
      AN    M 3.1;
      );
      A     M 7.0;
      A     M 7.1;
      A     M 7.2;
      A     M 3.0;
      A     M 0.1;
      L     DB30.DBW 118;
      SD    T 1;
NETWORK
TITLE =
      A     DB50.DBX 1.3;
      L     DB30.DBW 120;
      SD    T 2;
NETWORK
TITLE =
      A     M 21.4;
      A     M 0.1;
      L     DB30.DBW 122;
      SD    T 3;
NETWORK
TITLE =
      A     M 21.3;
      A     DB50.DBX 1.5;
      A     DB50.DBX 1.2;
      A     M 0.1;
      L     DB30.DBW 124;
      SD    T 4;
NETWORK
TITLE =
      A     M 21.7;
      AN    DB50.DBX 1.5;
      A     M 0.1;
      L     DB30.DBW 126;
      SD    T 5;
NETWORK
TITLE =
      A     M 21.6;
      AN    DB50.DBX 2.3;
      A(;
      O     M 0.1;
      O     M 42.0;
      );
      L     DB30.DBW 128;
      SD    T 6;
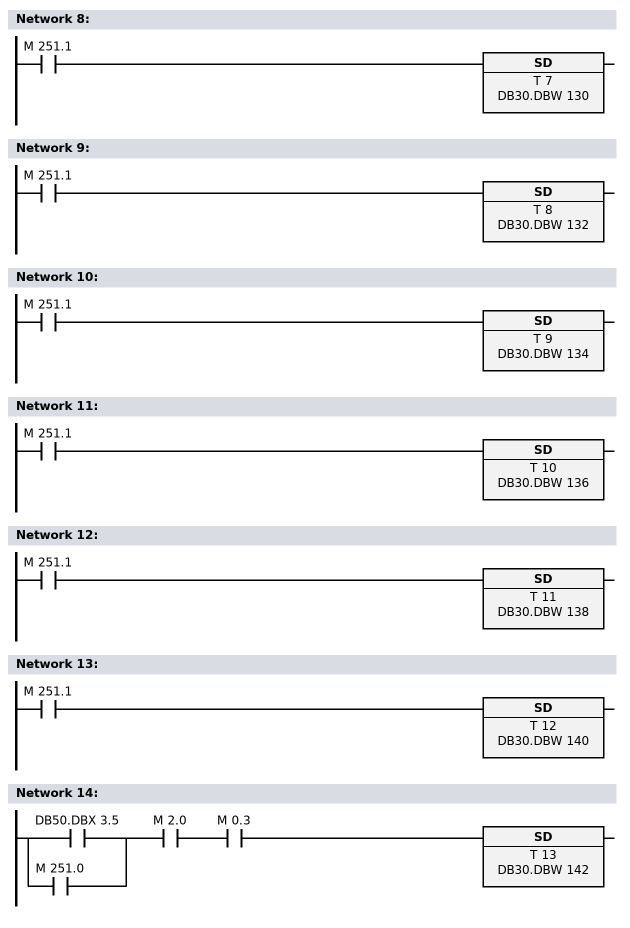
NETWORK
TITLE =
      A     M 251.1;
      L     DB30.DBW 130;
      SD    T 7;
NETWORK
TITLE =
      A     M 251.1;
      L     DB30.DBW 132;
      SD    T 8;
NETWORK
TITLE =
      A     M 251.1;
      L     DB30.DBW 134;
      SD    T 9;
NETWORK
TITLE =
      A     M 251.1;
      L     DB30.DBW 136;
      SD    T 10;
NETWORK
TITLE =
      A     M 251.1;
      L     DB30.DBW 138;
      SD    T 11;
NETWORK
TITLE =
      A     M 251.1;
      L     DB30.DBW 140;
      SD    T 12;
NETWORK
TITLE =
      A(;
      O     DB50.DBX 3.5;
      O     M 251.0;
      );
      A     M 2.0;
      A     M 0.3;
      L     DB30.DBW 142;
      SD    T 13;
END_FUNCTION

FUNCTION FC 19 : VOID
VERSION : 0.1
BEGIN
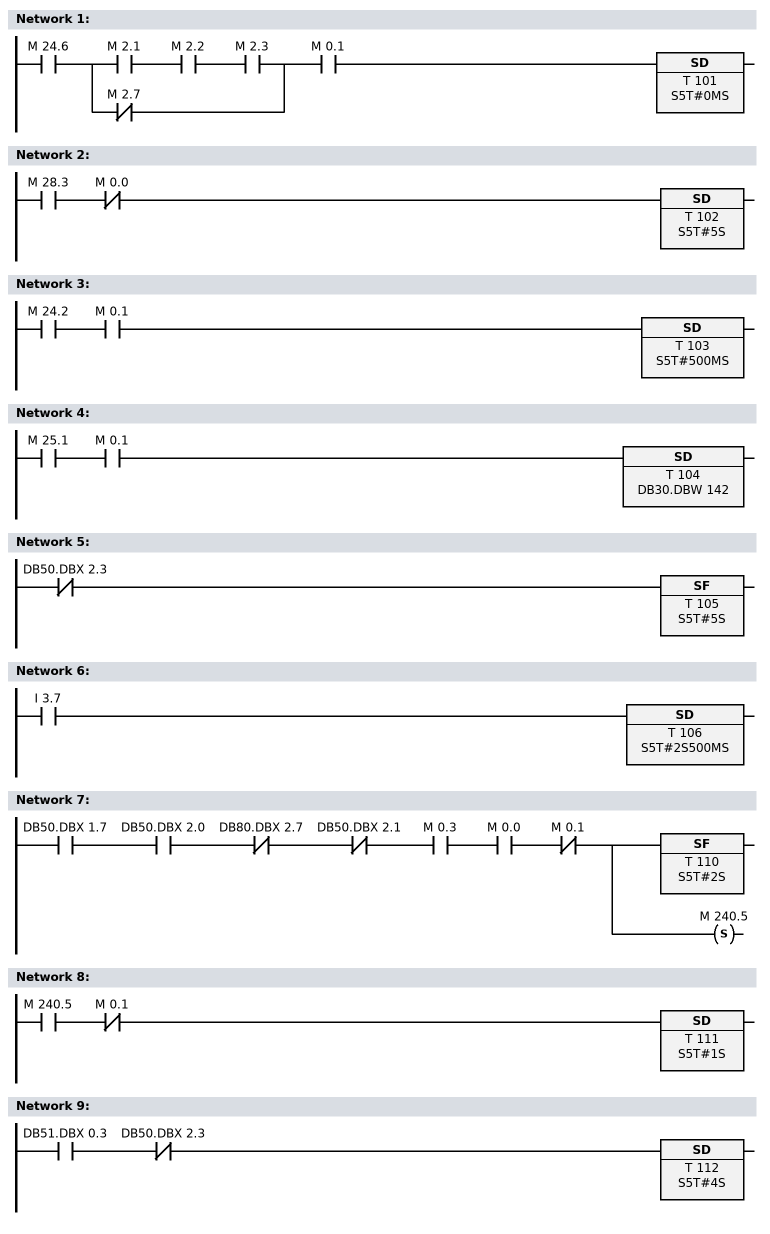
NETWORK
TITLE =
      A     M 24.6;
      A(;
      A     M 2.1;
      A     M 2.2;
      A     M 2.3;
      ON    M 2.7;
      );
      A     M 0.1;
      L     S5T#0MS;
      SD    T 101;
NETWORK
TITLE =
      A     M 28.3;
      AN    M 0.0;
      L     S5T#5S;
      SD    T 102;
NETWORK
TITLE =
      A     M 24.2;
      A     M 0.1;
      L     S5T#500MS;
      SD    T 103;
NETWORK
TITLE =
      A     M 25.1;
      A     M 0.1;
      L     DB30.DBW 142;
      SD    T 104;
NETWORK
TITLE =
      AN    DB50.DBX 2.3;
      L     S5T#5S;
      SF    T 105;
NETWORK
TITLE =
      A     I 3.7;
      L     S5T#2S500MS;
      SD    T 106;
NETWORK
TITLE =
      A     DB50.DBX 1.7;
      A     DB50.DBX 2.0;
      AN    DB80.DBX 2.7;
      AN    DB50.DBX 2.1;
      A     M 0.3;
      A     M 0.0;
      AN    M 0.1;
      L     S5T#2S;
      SF    T 110;
      S     M 240.5;
NETWORK
TITLE =
      A     M 240.5;
      AN    M 0.1;
      L     S5T#1S;
      SD    T 111;
NETWORK
TITLE =
      A     DB51.DBX 0.3;
      AN    DB50.DBX 2.3;
      L     S5T#4S;
      SD    T 112;
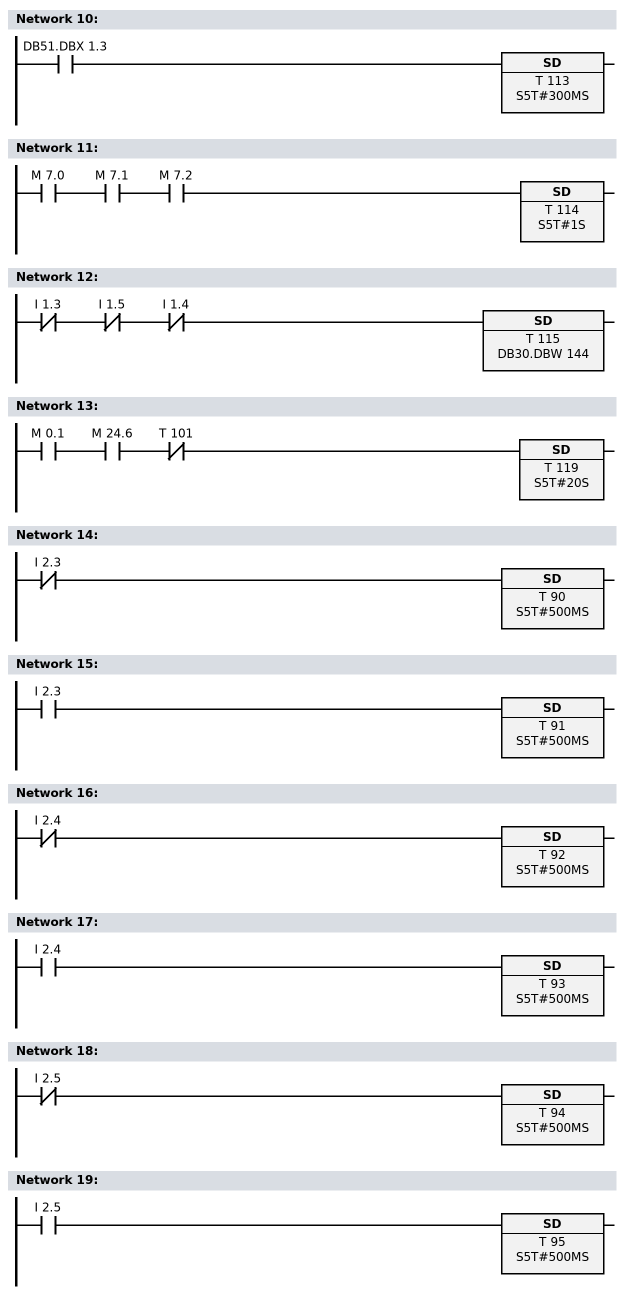
NETWORK
TITLE =
      A     DB51.DBX 1.3;
      L     S5T#300MS;
      SD    T 113;
NETWORK
TITLE =
      A     M 7.0;
      A     M 7.1;
      A     M 7.2;
      L     S5T#1S;
      SD    T 114;
NETWORK
TITLE =
      AN    I 1.3;
      AN    I 1.5;
      AN    I 1.4;
      L     DB30.DBW 144;
      SD    T 115;
NETWORK
TITLE =
      A     M 0.1;
      A     M 24.6;
      AN    T 101;
      L     S5T#20S;
      SD    T 119;
NETWORK
TITLE =
      AN    I 2.3;
      L     S5T#500MS;
      SD    T 90;
NETWORK
TITLE =
      A     I 2.3;
      L     S5T#500MS;
      SD    T 91;
NETWORK
TITLE =
      AN    I 2.4;
      L     S5T#500MS;
      SD    T 92;
NETWORK
TITLE =
      A     I 2.4;
      L     S5T#500MS;
      SD    T 93;
NETWORK
TITLE =
      AN    I 2.5;
      L     S5T#500MS;
      SD    T 94;
NETWORK
TITLE =
      A     I 2.5;
      L     S5T#500MS;
      SD    T 95;
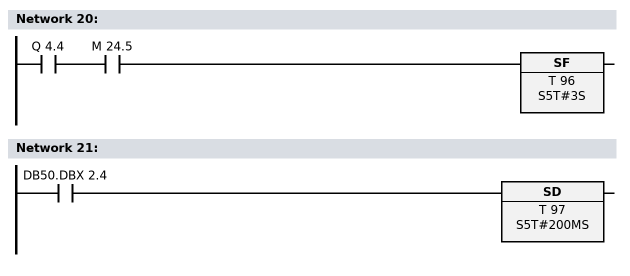
NETWORK
TITLE =
      A     Q 4.4;
      A     M 24.5;
      L     S5T#3S;
      SF    T 96;
NETWORK
TITLE =
      A     DB50.DBX 2.4;
      L     S5T#200MS;
      SD    T 97;
NETWORK
TITLE =
NETWORK
TITLE =
NETWORK
TITLE =
END_FUNCTION

FUNCTION FC 20 : VOID
VERSION : 0.1
BEGIN
// (block stored without names or comments; labels and parameter names are numbered)
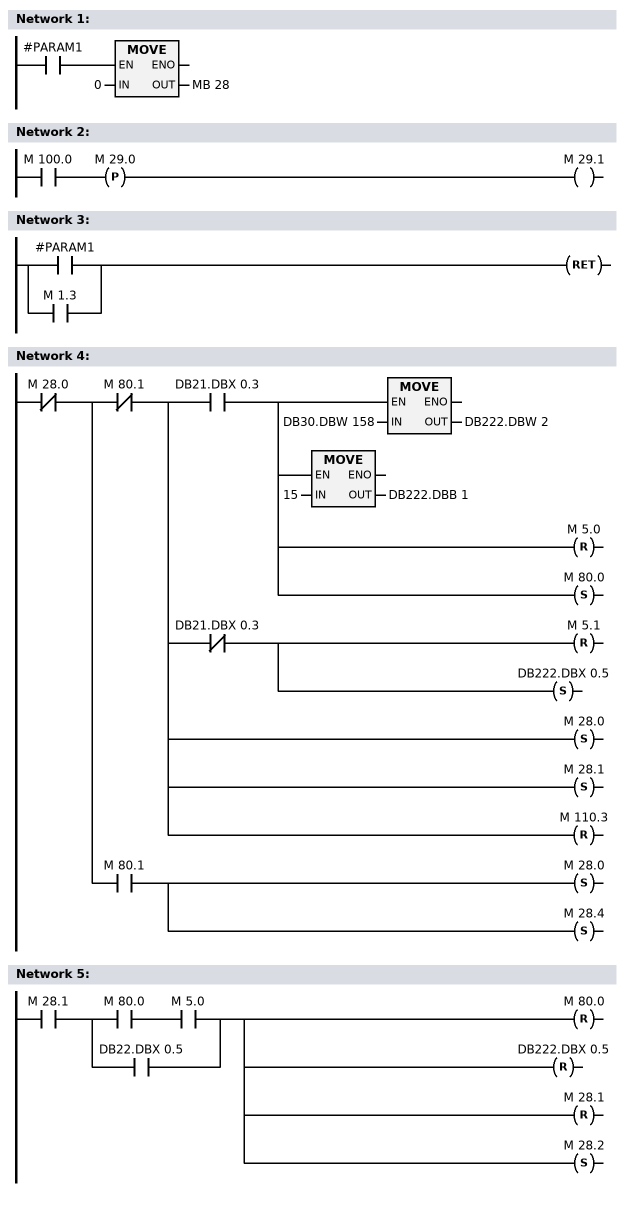
NETWORK
TITLE =
      A     #PARAM1;
      JNB   M001;
      L     0;
      T     MB 28;
M001: NOP   0;
NETWORK
TITLE =
      A     M 100.0;
      FP    M 29.0;
      =     M 29.1;
NETWORK
TITLE =
      O     #PARAM1;
      O     M 1.3;
      BEC;
NETWORK
TITLE =
      AN    M 28.0;
      =     L 0.0;
      A     L 0.0;
      AN    M 80.1;
      =     L 0.1;
      A     L 0.1;
      A     DB21.DBX 0.3;
      =     L 0.2;
      A     L 0.2;
      JNB   M002;
      L     DB30.DBW 158;
      T     DB222.DBW 2;
M002: NOP   0;
      A     L 0.2;
      JNB   M003;
      L     15;
      T     DB222.DBB 1;
M003: NOP   0;
      A     L 0.2;
      BLD   102;
      R     M 5.0;
      A     L 0.2;
      BLD   102;
      S     M 80.0;
      A     L 0.1;
      AN    DB21.DBX 0.3;
      R     M 5.1;
      S     DB222.DBX 0.5;
      A     L 0.1;
      BLD   102;
      S     M 28.0;
      A     L 0.1;
      BLD   102;
      S     M 28.1;
      A     L 0.1;
      BLD   102;
      R     M 110.3;
      A     L 0.0;
      A     M 80.1;
      S     M 28.0;
      S     M 28.4;
NETWORK
TITLE =
      A     M 28.1;
      A(;
      A     M 80.0;
      A     M 5.0;
      O     DB22.DBX 0.5;
      );
      R     M 80.0;
      R     DB222.DBX 0.5;
      R     M 28.1;
      S     M 28.2;
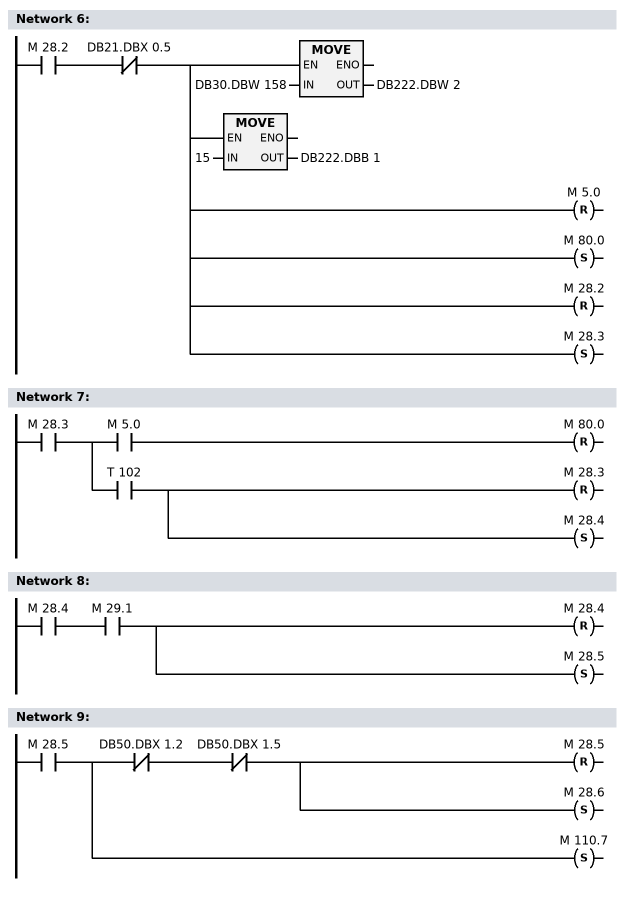
NETWORK
TITLE =
      A     M 28.2;
      AN    DB21.DBX 0.5;
      =     L 0.0;
      A     L 0.0;
      JNB   M004;
      L     DB30.DBW 158;
      T     DB222.DBW 2;
M004: NOP   0;
      A     L 0.0;
      JNB   M005;
      L     15;
      T     DB222.DBB 1;
M005: NOP   0;
      A     L 0.0;
      BLD   102;
      R     M 5.0;
      A     L 0.0;
      BLD   102;
      S     M 80.0;
      A     L 0.0;
      BLD   102;
      R     M 28.2;
      A     L 0.0;
      BLD   102;
      S     M 28.3;
NETWORK
TITLE =
      A     M 28.3;
      =     L 0.0;
      A     L 0.0;
      A     M 5.0;
      R     M 80.0;
      A     L 0.0;
      A     T 102;
      R     M 28.3;
      S     M 28.4;
NETWORK
TITLE =
      A     M 28.4;
      A     M 29.1;
      R     M 28.4;
      S     M 28.5;
NETWORK
TITLE =
      A     M 28.5;
      =     L 0.0;
      A     L 0.0;
      AN    DB50.DBX 1.2;
      AN    DB50.DBX 1.5;
      R     M 28.5;
      S     M 28.6;
      A     L 0.0;
      BLD   102;
      S     M 110.7;
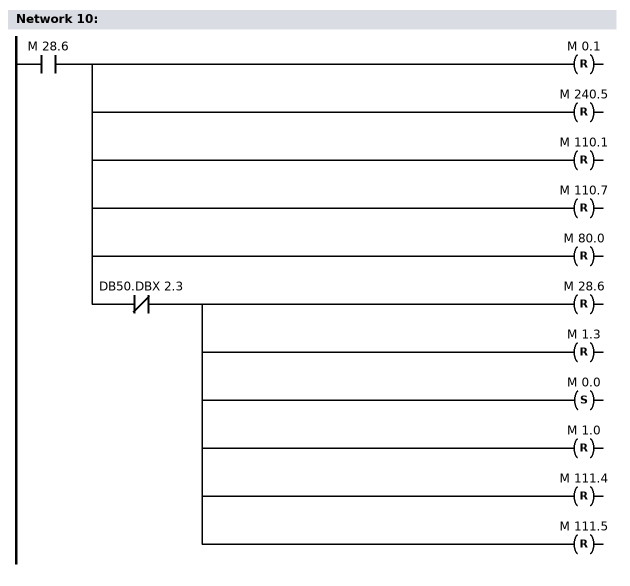
NETWORK
TITLE =
      A     M 28.6;
      =     L 0.0;
      A     L 0.0;
      BLD   102;
      R     M 0.1;
      A     L 0.0;
      BLD   102;
      R     M 240.5;
      A     L 0.0;
      BLD   102;
      R     M 110.1;
      A     L 0.0;
      BLD   102;
      R     M 110.7;
      A     L 0.0;
      BLD   102;
      R     M 80.0;
      A     L 0.0;
      AN    DB50.DBX 2.3;
      R     M 28.6;
      R     M 1.3;
      S     M 0.0;
      R     M 1.0;
      R     M 111.4;
      R     M 111.5;
END_FUNCTION

FUNCTION FC 21 : VOID
VERSION : 0.1
BEGIN
// (block stored without names or comments; labels and parameter names are numbered)
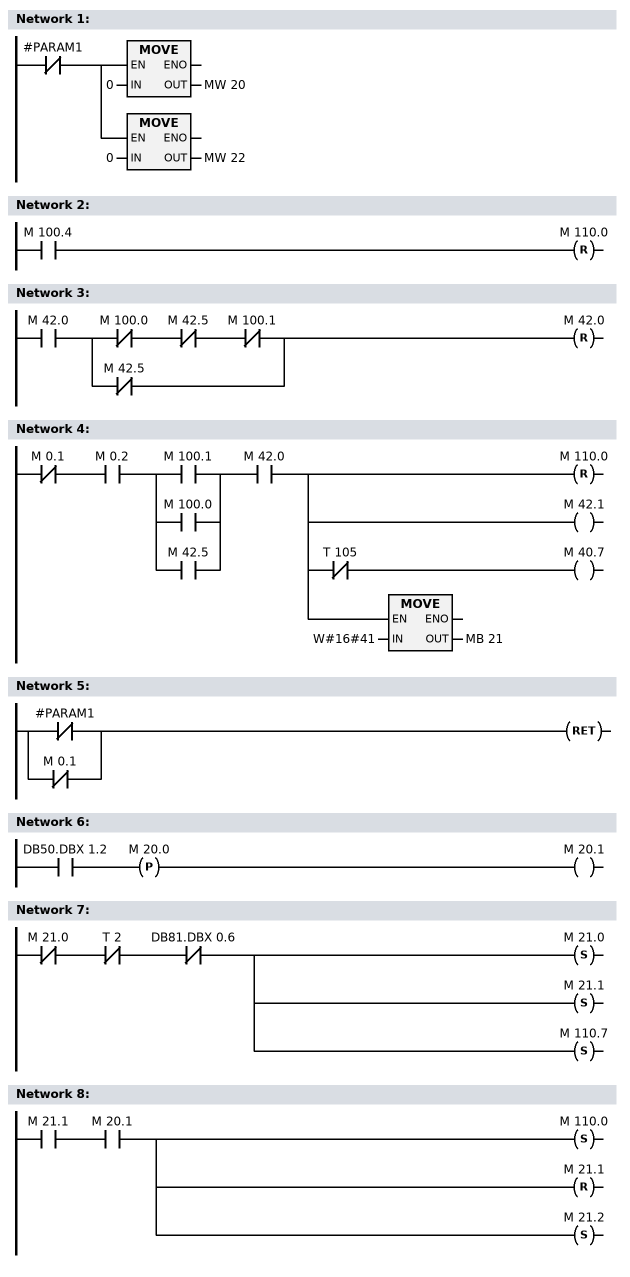
NETWORK
TITLE =
      AN    #PARAM1;
      =     L 0.0;
      A     L 0.0;
      JNB   M001;
      L     0;
      T     MW 20;
M001: NOP   0;
      A     L 0.0;
      JNB   M002;
      L     0;
      T     MW 22;
M002: NOP   0;
NETWORK
TITLE =
      A     M 100.4;
      R     M 110.0;
NETWORK
TITLE =
      A     M 42.0;
      A(;
      AN    M 100.0;
      AN    M 42.5;
      AN    M 100.1;
      ON    M 42.5;
      );
      R     M 42.0;
NETWORK
TITLE =
      AN    M 0.1;
      A     M 0.2;
      A(;
      O     M 100.1;
      O     M 100.0;
      O     M 42.5;
      );
      A     M 42.0;
      =     L 0.0;
      A     L 0.0;
      BLD   102;
      R     M 110.0;
      A     L 0.0;
      BLD   102;
      =     M 42.1;
      A     L 0.0;
      AN    T 105;
      =     M 40.7;
      A     L 0.0;
      JNB   M003;
      L     W#16#41;
      T     MB 21;
M003: NOP   0;
NETWORK
TITLE =
      AN    #PARAM1;
      ON    M 0.1;
      BEC;
NETWORK
TITLE =
      A     DB50.DBX 1.2;
      FP    M 20.0;
      =     M 20.1;
NETWORK
TITLE =
      AN    M 21.0;
      AN    T 2;
      AN    DB81.DBX 0.6;
      S     M 21.0;
      S     M 21.1;
      S     M 110.7;
NETWORK
TITLE =
      A     M 21.1;
      A     M 20.1;
      S     M 110.0;
      R     M 21.1;
      S     M 21.2;
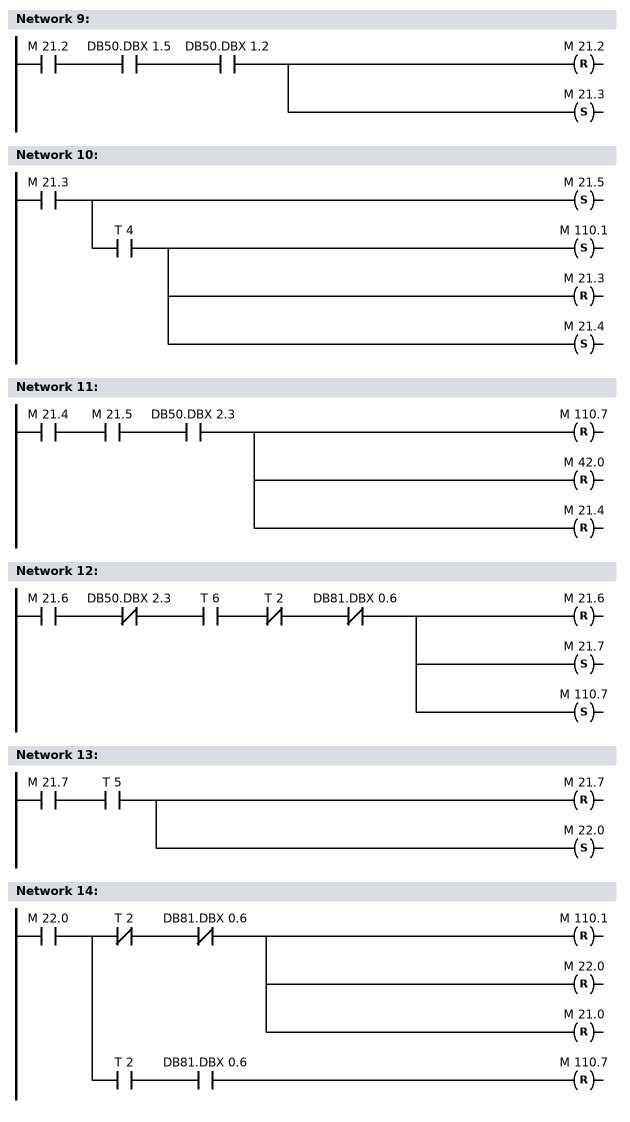
NETWORK
TITLE =
      A     M 21.2;
      A     DB50.DBX 1.5;
      A     DB50.DBX 1.2;
      R     M 21.2;
      S     M 21.3;
NETWORK
TITLE =
      A     M 21.3;
      =     L 0.0;
      A     L 0.0;
      BLD   102;
      S     M 21.5;
      A     L 0.0;
      A     T 4;
      S     M 110.1;
      R     M 21.3;
      S     M 21.4;
NETWORK
TITLE =
      A     M 21.4;
      A     M 21.5;
      A     DB50.DBX 2.3;
      R     M 110.7;
      R     M 42.0;
      R     M 21.4;
NETWORK
TITLE =
      A     M 21.6;
      AN    DB50.DBX 2.3;
      A     T 6;
      AN    T 2;
      AN    DB81.DBX 0.6;
      R     M 21.6;
      S     M 21.7;
      S     M 110.7;
NETWORK
TITLE =
      A     M 21.7;
      A     T 5;
      R     M 21.7;
      S     M 22.0;
NETWORK
TITLE =
      A     M 22.0;
      =     L 0.0;
      A     L 0.0;
      AN    T 2;
      AN    DB81.DBX 0.6;
      R     M 110.1;
      R     M 22.0;
      R     M 21.0;
      A     L 0.0;
      A     T 2;
      A     DB81.DBX 0.6;
      R     M 110.7;
END_FUNCTION

FUNCTION FC 22 : VOID
VERSION : 0.1
BEGIN
// (block stored without names or comments; labels and parameter names are numbered)
NETWORK
TITLE =
      AN    #PARAM1;
      JNB   M001;
      L     0;
      T     MW 24;
      T     MB 26;
M001: NOP   0;
NETWORK
TITLE =
      AN    #PARAM1;
      BEC;
NETWORK
TITLE =
      A     M 24.0;
      JC    M002;
      L     DB30.DBW 154;
      T     DB222.DBW 2;
      L     18;
      T     DB222.DBB 1;
      L     0;
      T     MW 10;
      L     0;
      T     MW 12;
      L     0;
      T     MW 14;
      R     M 2.1;
      R     M 2.2;
      R     M 2.3;
      R     M 5.0;
      AN    DB21.DBX 0.5;
      S     M 80.0;
      S     M 24.0;
      S     M 24.1;
M002: NOP   0;
NETWORK
TITLE =
      AN    M 24.1;
      JC    M003;
      A     M 5.0;
      R     M 80.0;
      R     M 23.0;
      R     M 24.1;
      S     M 24.2;
M003: NOP   0;
NETWORK
TITLE =
      AN    M 24.2;
      JC    M004;
      S     M 110.3;
      A     T 103;
      S     M 111.5;
      S     M 111.4;
      R     M 24.2;
      S     M 24.3;
M004: NOP   0;
NETWORK
TITLE =
      AN    M 24.3;
      JC    M005;
      A     M 1.6;
      O     T 1;
      R     M 24.3;
      S     M 24.4;
M005: NOP   0;
NETWORK
TITLE =
      AN    M 24.4;
      JC    M006;
      L     DB30.DBW 156;
      T     DB222.DBW 2;
      L     DB30.DBW 162;
      T     DB222.DBB 1;
      R     M 5.0;
      AN    DB21.DBX 0.5;
      R     M 24.4;
      S     M 24.5;
M006: NOP   0;
NETWORK
TITLE =
      AN    M 24.5;
      JC    M007;
      S     M 80.0;
      A     M 5.0;
      R     M 24.5;
      S     M 24.6;
M007: NOP   0;
NETWORK
TITLE =
      AN    M 24.6;
      JC    M008;
      R     M 80.0;
      A     T 101;
      R     M 111.5;
      R     M 110.3;
      S     M 23.0;
      R     M 24.6;
      S     M 24.7;
M008: NOP   0;
NETWORK
TITLE =
      AN    M 24.7;
      JC    M009;
      L     DB30.DBW 158;
      T     DB222.DBW 2;
      L     DB30.DBW 164;
      T     DB222.DBB 1;
      R     M 5.0;
      AN    DB21.DBX 0.5;
      R     M 24.7;
      S     M 25.0;
M009: NOP   0;
NETWORK
TITLE =
      AN    M 25.0;
      JC    M010;
      S     M 80.0;
      A     M 5.0;
      R     M 25.0;
      S     M 25.1;
M010: NOP   0;
NETWORK
TITLE =
      AN    M 25.1;
      JC    M011;
      R     M 80.0;
      A     T 104;
      R     M 111.4;
      S     M 25.2;
      R     M 25.1;
M011: NOP   0;
NETWORK
TITLE =
      AN    M 25.3;
      JC    M012;
      L     DB30.DBW 160;
      T     DB222.DBW 2;
      L     DB30.DBW 164;
      T     DB222.DBB 1;
      R     M 5.0;
      AN    DB21.DBX 0.5;
      R     M 25.3;
      S     M 25.4;
M012: NOP   0;
NETWORK
TITLE =
      AN    M 25.4;
      JC    M013;
      S     M 80.0;
      A     M 5.0;
      R     M 80.0;
      R     M 25.4;
M013: NOP   0;
END_FUNCTION

FUNCTION FC 30 : VOID
VERSION : 0.1
BEGIN
// (block stored without names or comments; labels and parameter names are numbered)
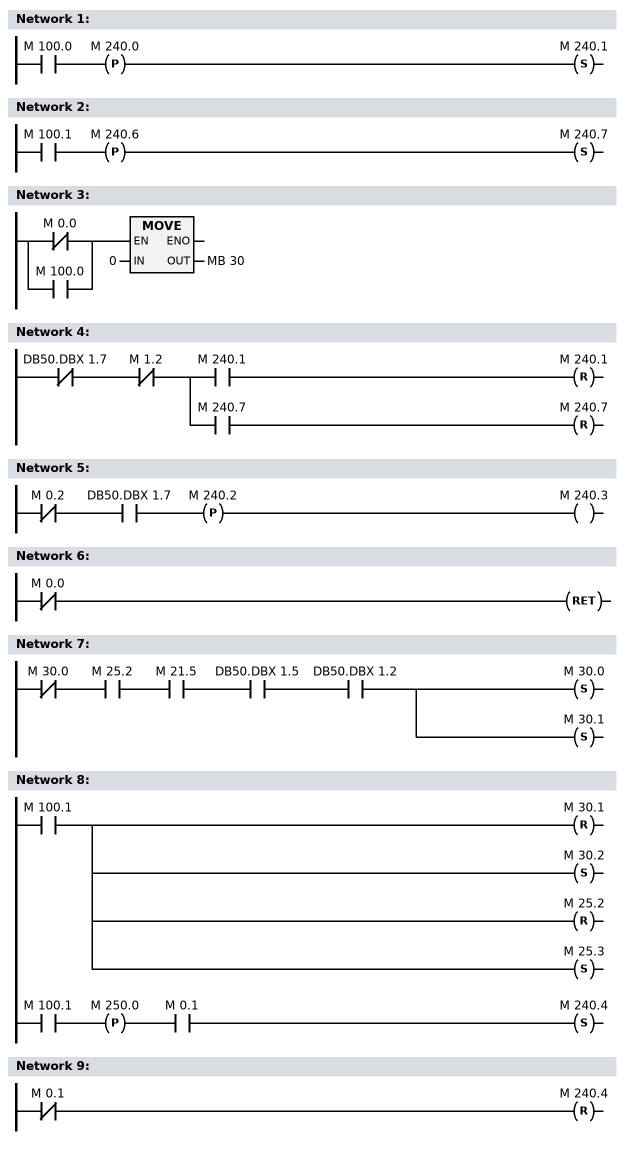
NETWORK
TITLE =
      A     M 100.0;
      FP    M 240.0;
      S     M 240.1;
NETWORK
TITLE =
      A     M 100.1;
      FP    M 240.6;
      S     M 240.7;
NETWORK
TITLE =
      A(;
      ON    M 0.0;
      O     M 100.0;
      );
      JNB   M001;
      L     0;
      T     MB 30;
M001: NOP   0;
NETWORK
TITLE =
      AN    DB50.DBX 1.7;
      AN    M 1.2;
      =     L 0.0;
      A     L 0.0;
      A     M 240.1;
      R     M 240.1;
      A     L 0.0;
      A     M 240.7;
      R     M 240.7;
NETWORK
TITLE =
      AN    M 0.2;
      A     DB50.DBX 1.7;
      FP    M 240.2;
      =     M 240.3;
NETWORK
TITLE =
      AN    M 0.0;
      BEC;
NETWORK
TITLE =
      AN    M 30.0;
      A     M 25.2;
      A     M 21.5;
      A     DB50.DBX 1.5;
      A     DB50.DBX 1.2;
      S     M 30.0;
      S     M 30.1;
NETWORK
TITLE =
      A     M 100.1;
      =     L 0.0;
      A     L 0.0;
      BLD   102;
      R     M 30.1;
      A     L 0.0;
      BLD   102;
      S     M 30.2;
      A     L 0.0;
      BLD   102;
      R     M 25.2;
      A     L 0.0;
      BLD   102;
      S     M 25.3;
      A(;
      A     L 0.0;
      FP    M 250.0;
      );
      A     M 0.1;
      S     M 240.4;
NETWORK
TITLE =
      AN    M 0.1;
      R     M 240.4;
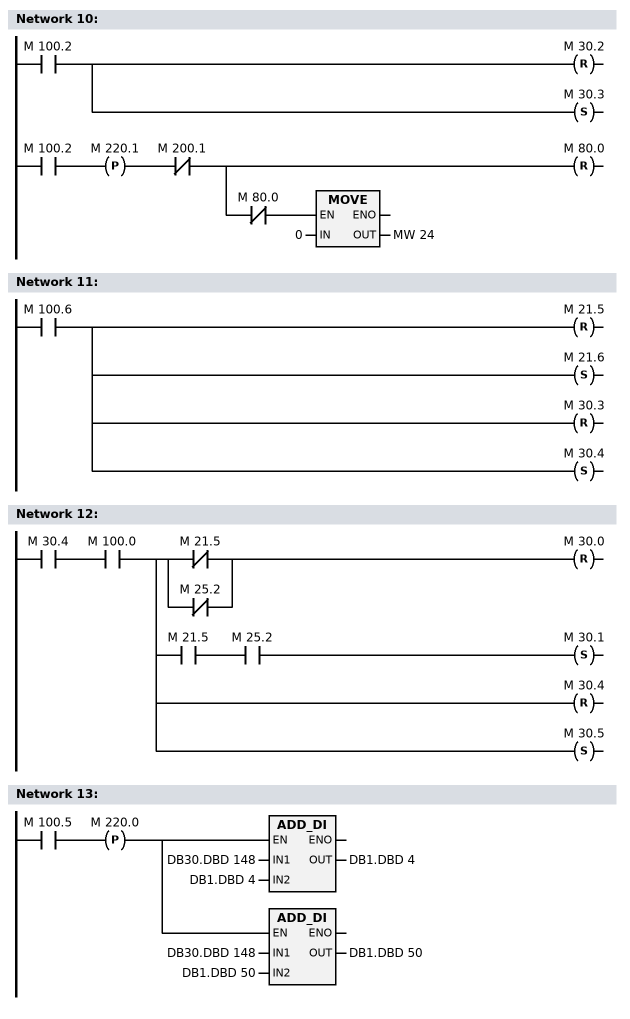
NETWORK
TITLE =
      A     M 100.2;
      =     L 0.0;
      A     L 0.0;
      BLD   102;
      R     M 30.2;
      A     L 0.0;
      BLD   102;
      S     M 30.3;
      A(;
      A     L 0.0;
      FP    M 220.1;
      );
      AN    M 200.1;
      =     L 0.1;
      A     L 0.1;
      BLD   102;
      R     M 80.0;
      A     L 0.1;
      AN    M 80.0;
      JNB   M002;
      L     0;
      T     MW 24;
M002: NOP   0;
NETWORK
TITLE =
      A     M 100.6;
      R     M 21.5;
      S     M 21.6;
      R     M 30.3;
      S     M 30.4;
NETWORK
TITLE =
      A     M 30.4;
      A     M 100.0;
      =     L 0.0;
      A     L 0.0;
      A(;
      ON    M 21.5;
      ON    M 25.2;
      );
      R     M 30.0;
      A     L 0.0;
      A     M 21.5;
      A     M 25.2;
      S     M 30.1;
      A     L 0.0;
      BLD   102;
      R     M 30.4;
      A     L 0.0;
      BLD   102;
      S     M 30.5;
NETWORK
TITLE =
      A     M 100.5;
      FP    M 220.0;
      =     L 0.0;
      A     L 0.0;
      JNB   M003;
      L     DB30.DBD 148;
      L     DB1.DBD 4;
      +D;
      T     DB1.DBD 4;
M003: NOP   0;
      A     L 0.0;
      JNB   M004;
      L     DB30.DBD 148;
      L     DB1.DBD 50;
      +D;
      T     DB1.DBD 50;
M004: NOP   0;
END_FUNCTION

FUNCTION FC 59 : VOID
VERSION : 0.1
BEGIN
// (block stored without names or comments; labels and parameter names are numbered)
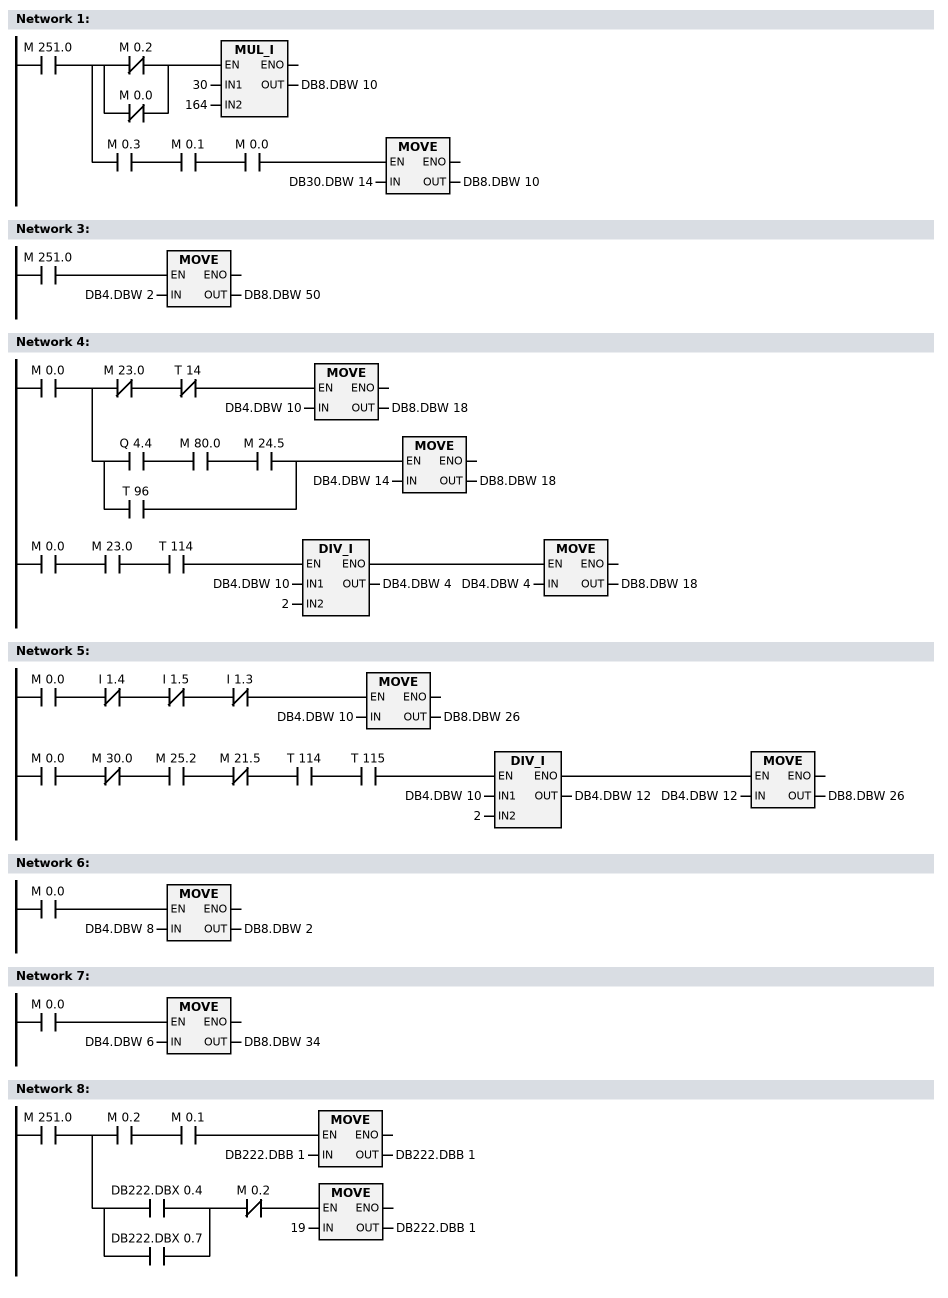
NETWORK
TITLE =
      A     M 251.0;
      =     L 12.0;
      A     L 12.0;
      A(;
      ON    M 0.2;
      ON    M 0.0;
      );
      JNB   M001;
      L     30;
      L     164;
      *I;
      T     DB8.DBW 10;
M001: NOP   0;
      A     L 12.0;
      A     M 0.3;
      A     M 0.1;
      A     M 0.0;
      JNB   M002;
      L     DB30.DBW 14;
      T     DB8.DBW 10;
M002: NOP   0;
NETWORK
TITLE =
      A     M 0.0;
      =     L 12.0;
      A     L 12.0;
      A     M 251.1;
      =     L 12.1;
      A     L 12.1;
      A(;
      L     DB30.DBW 12;
      L     400;
      >=I;
      );
      JNB   M003;
      L     DB4.DBW 2;
      T     DB8.DBW 42;
M003: NOP   0;
      A(;
      A     L 12.1;
      A(;
      L     DB30.DBW 12;
      L     400;
      <=I;
      );
      JNB   M004;
      L     DB4.DBW 2;
      L     3;
      /I;
      T     DB1.DBW 32;
      AN    OV;
      SAVE;
      CLR;
M004: A     BR;
      );
      JNB   M005;
      L     DB1.DBW 32;
      T     DB8.DBW 42;
M005: NOP   0;
      A     L 12.0;
      JNB   M006;
      L     DB4.DBW 2;
      T     DB8.DBW 42;
M006: NOP   0;
NETWORK
TITLE =
      A     M 251.0;
      JNB   M007;
      L     DB4.DBW 2;
      T     DB8.DBW 50;
M007: NOP   0;
NETWORK
TITLE =
      A     M 0.0;
      =     L 12.0;
      A     L 12.0;
      AN    M 23.0;
      AN    T 14;
      JNB   M008;
      L     DB4.DBW 10;
      T     DB8.DBW 18;
M008: NOP   0;
      A(;
      A     L 12.0;
      A     M 23.0;
      A     T 114;
      JNB   M009;
      L     DB4.DBW 10;
      L     2;
      /I;
      T     DB4.DBW 4;
      AN    OV;
      SAVE;
      CLR;
M009: A     BR;
      );
      JNB   M010;
      L     DB4.DBW 4;
      T     DB8.DBW 18;
M010: NOP   0;
      A     L 12.0;
      A(;
      A     Q 4.4;
      A     M 80.0;
      A     M 24.5;
      O     T 96;
      );
      JNB   M011;
      L     DB4.DBW 14;
      T     DB8.DBW 18;
M011: NOP   0;
NETWORK
TITLE =
      A     M 0.0;
      =     L 12.0;
      A     L 12.0;
      AN    I 1.4;
      AN    I 1.5;
      AN    I 1.3;
      JNB   M012;
      L     DB4.DBW 10;
      T     DB8.DBW 26;
M012: NOP   0;
      A(;
      A     L 12.0;
      AN    M 30.0;
      A     M 25.2;
      AN    M 21.5;
      A     T 114;
      A     T 115;
      JNB   M013;
      L     DB4.DBW 10;
      L     2;
      /I;
      T     DB4.DBW 12;
      AN    OV;
      SAVE;
      CLR;
M013: A     BR;
      );
      JNB   M014;
      L     DB4.DBW 12;
      T     DB8.DBW 26;
M014: NOP   0;
NETWORK
TITLE =
      A     M 0.0;
      JNB   M015;
      L     DB4.DBW 8;
      T     DB8.DBW 2;
M015: NOP   0;
NETWORK
TITLE =
      A     M 0.0;
      JNB   M016;
      L     DB4.DBW 6;
      T     DB8.DBW 34;
M016: NOP   0;
NETWORK
TITLE =
      A     M 251.0;
      =     L 12.0;
      A     L 12.0;
      A     M 0.2;
      A     M 0.1;
      JNB   M017;
      L     DB222.DBB 1;
      T     DB222.DBB 1;
M017: NOP   0;
      A     L 12.0;
      A(;
      O     DB222.DBX 0.4;
      O     DB222.DBX 0.7;
      );
      AN    M 0.2;
      JNB   M018;
      L     19;
      T     DB222.DBB 1;
M018: NOP   0;
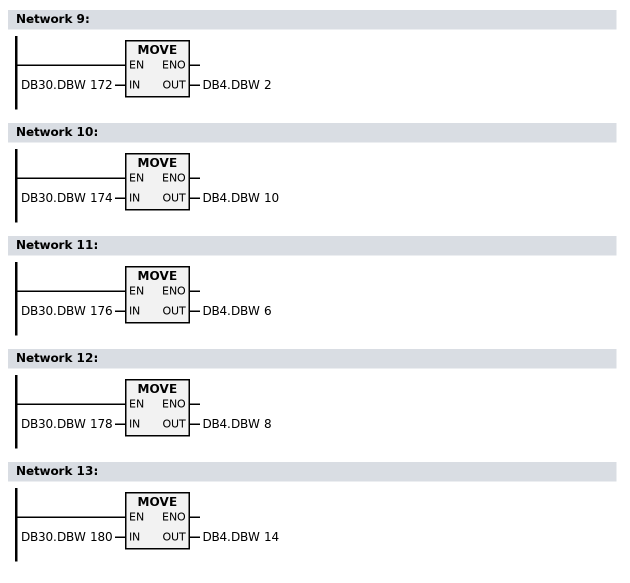
NETWORK
TITLE =
      L     DB30.DBW 172;
      T     DB4.DBW 2;
NETWORK
TITLE =
      L     DB30.DBW 174;
      T     DB4.DBW 10;
NETWORK
TITLE =
      L     DB30.DBW 176;
      T     DB4.DBW 6;
NETWORK
TITLE =
      L     DB30.DBW 178;
      T     DB4.DBW 8;
NETWORK
TITLE =
      L     DB30.DBW 180;
      T     DB4.DBW 14;
END_FUNCTION

FUNCTION FC 60 : VOID
VERSION : 0.1
BEGIN
// (block stored without names or comments; labels and parameter names are numbered)
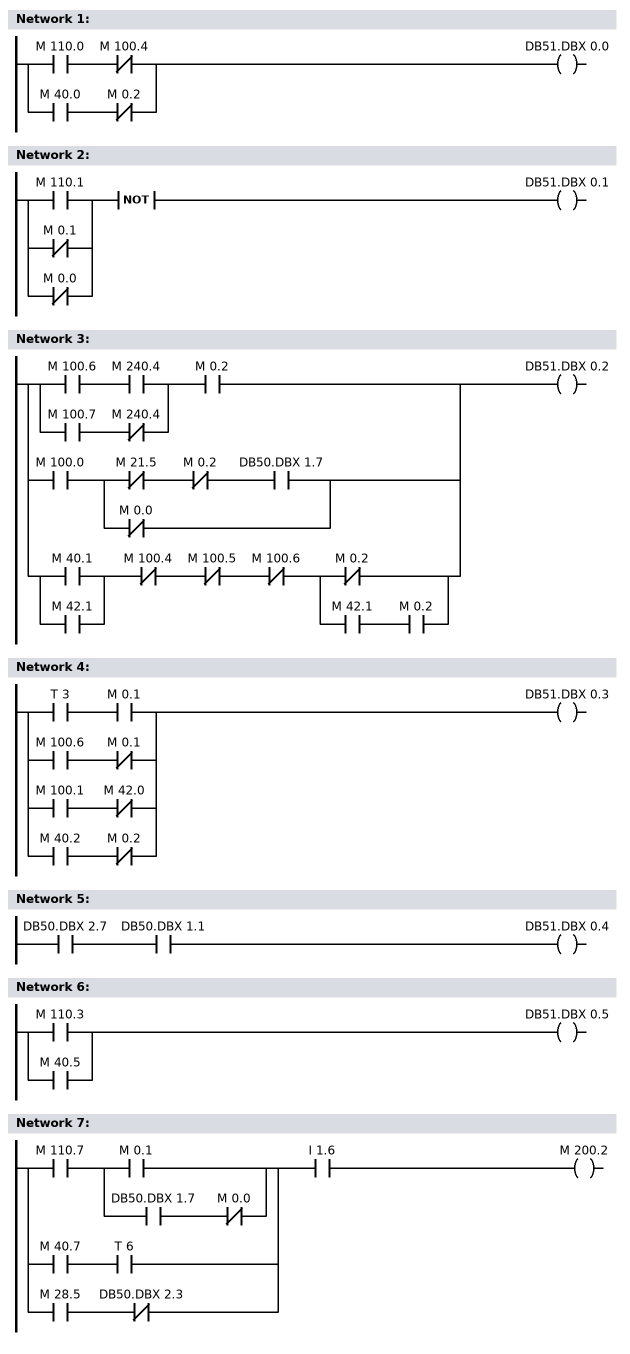
NETWORK
TITLE =
      A     M 110.0;
      AN    M 100.4;
      O;
      A     M 40.0;
      AN    M 0.2;
      =     DB51.DBX 0.0;
NETWORK
TITLE =
      A(;
      O     M 110.1;
      ON    M 0.1;
      ON    M 0.0;
      );
      NOT;
      =     DB51.DBX 0.1;
NETWORK
TITLE =
      A(;
      A     M 100.6;
      A     M 240.4;
      O;
      A     M 100.7;
      AN    M 240.4;
      );
      A     M 0.2;
      O;
      A     M 100.0;
      A(;
      AN    M 21.5;
      AN    M 0.2;
      A     DB50.DBX 1.7;
      ON    M 0.0;
      );
      O;
      A(;
      O     M 40.1;
      O     M 42.1;
      );
      AN    M 100.4;
      AN    M 100.5;
      AN    M 100.6;
      A(;
      ON    M 0.2;
      O;
      A     M 42.1;
      A     M 0.2;
      );
      =     DB51.DBX 0.2;
NETWORK
TITLE =
      A     T 3;
      A     M 0.1;
      O;
      A     M 100.6;
      AN    M 0.1;
      O;
      A     M 100.1;
      AN    M 42.0;
      O;
      A     M 40.2;
      AN    M 0.2;
      =     DB51.DBX 0.3;
NETWORK
TITLE =
      A     DB50.DBX 2.7;
      A     DB50.DBX 1.1;
      =     DB51.DBX 0.4;
NETWORK
TITLE =
      O     M 110.3;
      O     M 40.5;
      =     DB51.DBX 0.5;
NETWORK
TITLE =
      A(;
      A     M 110.7;
      A(;
      O     M 0.1;
      O;
      A     DB50.DBX 1.7;
      AN    M 0.0;
      );
      O;
      A     M 40.7;
      A     T 6;
      O;
      A     M 28.5;
      AN    DB50.DBX 2.3;
      );
      A     I 1.6;
      =     M 200.2;
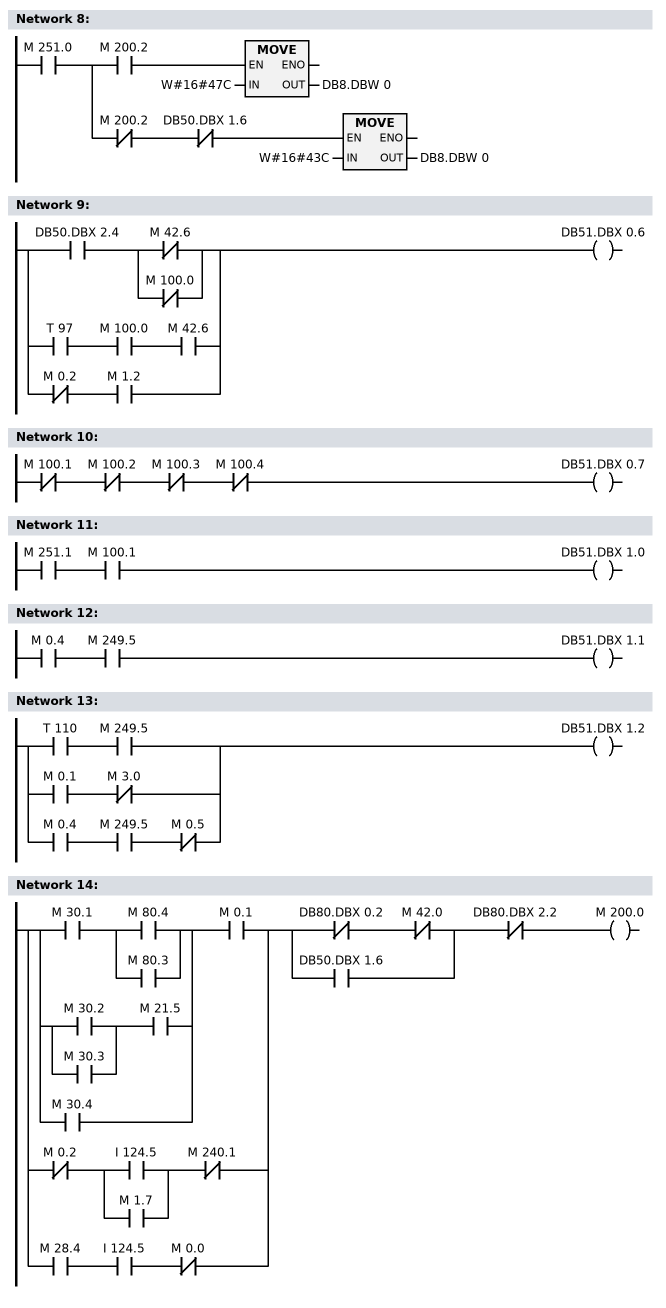
NETWORK
TITLE =
      A     M 251.0;
      =     L 0.0;
      A     L 0.0;
      A     M 200.2;
      JNB   M001;
      L     W#16#47C;
      T     DB8.DBW 0;
M001: NOP   0;
      A     L 0.0;
      AN    M 200.2;
      AN    DB50.DBX 1.6;
      JNB   M002;
      L     W#16#43C;
      T     DB8.DBW 0;
M002: NOP   0;
NETWORK
TITLE =
      A     DB50.DBX 2.4;
      A(;
      ON    M 42.6;
      ON    M 100.0;
      );
      O;
      A     T 97;
      A     M 100.0;
      A     M 42.6;
      O;
      AN    M 0.2;
      A     M 1.2;
      =     DB51.DBX 0.6;
NETWORK
TITLE =
      AN    M 100.1;
      AN    M 100.2;
      AN    M 100.3;
      AN    M 100.4;
      =     DB51.DBX 0.7;
NETWORK
TITLE =
      A     M 251.1;
      A     M 100.1;
      =     DB51.DBX 1.0;
NETWORK
TITLE =
      A     M 0.4;
      A     M 249.5;
      =     DB51.DBX 1.1;
NETWORK
TITLE =
      A     T 110;
      A     M 249.5;
      O;
      A     M 0.1;
      AN    M 3.0;
      O;
      A     M 0.4;
      A     M 249.5;
      AN    M 0.5;
      =     DB51.DBX 1.2;
NETWORK
TITLE =
      A(;
      A(;
      A     M 30.1;
      A(;
      O     M 80.4;
      O     M 80.3;
      );
      O;
      A(;
      O     M 30.2;
      O     M 30.3;
      );
      A     M 21.5;
      O     M 30.4;
      );
      A     M 0.1;
      O;
      AN    M 0.2;
      A(;
      O     I 124.5;
      O     M 1.7;
      );
      AN    M 240.1;
      O;
      A     M 28.4;
      A     I 124.5;
      AN    M 0.0;
      );
      A(;
      AN    DB80.DBX 0.2;
      AN    M 42.0;
      O     DB50.DBX 1.6;
      );
      AN    DB80.DBX 2.2;
      =     M 200.0;
